// ---- HMI/VISUs/Templates/Motors/GUI_TEMPLATE_NOTT_MOTOR_CONTROL.TcVIS
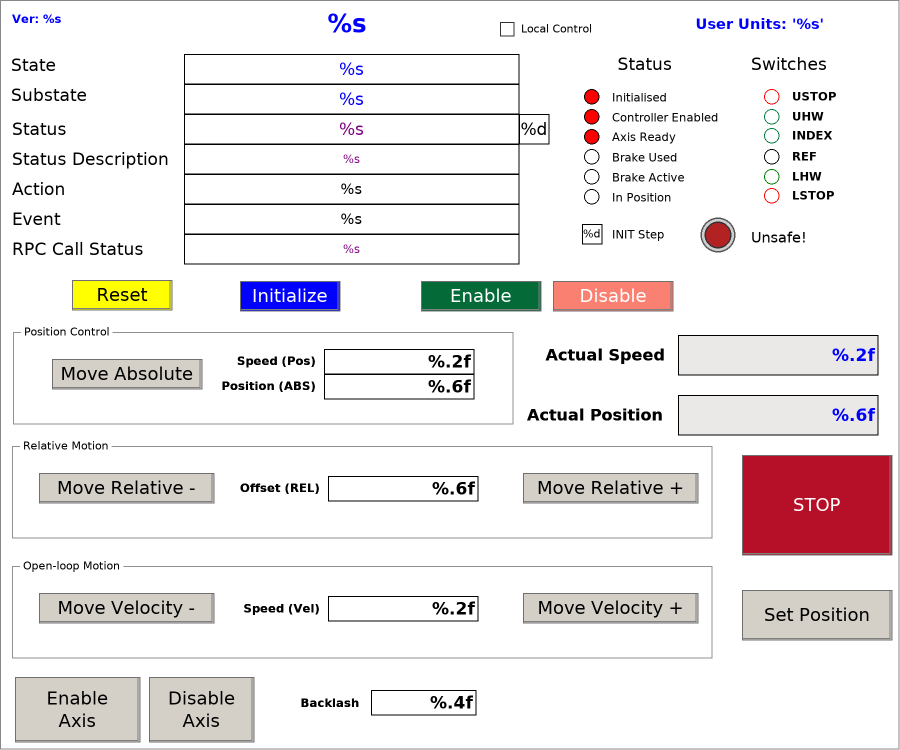
VISUALIZATION GUI_TEMPLATE_NOTT_MOTOR_CONTROL  // 900x750
VAR_IN_OUT
	m_Instance:	FB_NOTT_MOTOR;
END_VAR
VAR
	m_lrOffSet : LREAL := 0;
END_VAR
    GroupBox (12,558 700x100), "Open-loop Motion"
        Button (511,35 175x30), "Move Velocity +", input disabled if: NOT m_Instance.stat.bLocal OR NOT m_Instance.in_bSafe
            OnMouseDown: execute {
                m_Instance.ctrl.bLocalCmd := TRUE;
                m_Instance.ctrl.nCommand := E_MOTOR_COMMAND.MOTOR_MOVE;
                m_Instance.ctrl.nMoveType := E_MOTOR_MOVE_TYPE.VELOCITY;
                m_Instance.ctrl.nDirection := MC_Positive_Direction;
                m_Instance.ctrl.bExecute := TRUE;
            }
    Button (523,593 175x30), "Move Velocity +", input disabled if: NOT m_Instance.stat.bLocal OR NOT m_Instance.in_bSafe
        OnMouseDown: execute {
            m_Instance.ctrl.bLocalCmd := TRUE;
            m_Instance.ctrl.nCommand := E_MOTOR_COMMAND.MOTOR_MOVE;
            m_Instance.ctrl.nMoveType := E_MOTOR_MOVE_TYPE.VELOCITY;
            m_Instance.ctrl.nDirection := MC_Positive_Direction;
            m_Instance.ctrl.bExecute := TRUE;
        }
    GroupBox (12,438 700x100), "Relative Motion"
    GroupBox (13,324 500x100), "Position Control"
    Rectangle (184,54 335x30), "%s", text variable: m_Instance.stat.sState
    Rectangle (184,84 335x30), "%s", text variable: m_Instance.stat.sSubstate
    Button (72,280 100x30), "Reset", input disabled if: NOT m_Instance.stat.bLocal OR NOT m_Instance.in_bSafe
        OnMouseDown: execute {
            m_Instance.ctrl.bLocalCmd := TRUE;
            m_Instance.ctrl.nCommand := E_MOTOR_COMMAND.RESET;
            m_Instance.ctrl.bExecute := TRUE;
        }
    Button (240,281 100x30), "Initialize", input disabled if: NOT m_Instance.stat.bLocal OR NOT m_Instance.in_bSafe
        OnMouseDown: execute {
            m_Instance.ctrl.bLocalCmd := TRUE;
            m_Instance.ctrl.nCommand := E_MOTOR_COMMAND.INIT;
            m_Instance.ctrl.bExecute := TRUE;
        }
    Button (742,455 150x100), "STOP", input disabled if: NOT m_Instance.stat.bLocal OR NOT m_Instance.in_bSafe
        OnMouseDown: execute {
            m_Instance.ctrl.bLocalCmd := TRUE;
            m_Instance.ctrl.nCommand := E_MOTOR_COMMAND.STOP;
            m_Instance.ctrl.bExecute := TRUE;
        }
    Button (421,281 120x30), "Enable", input disabled if: NOT m_Instance.stat.bLocal OR NOT m_Instance.in_bSafe
        OnMouseDown: execute {
            m_Instance.ctrl.bLocalCmd := TRUE;
            m_Instance.ctrl.nCommand := E_MOTOR_COMMAND.ENABLE;
            m_Instance.ctrl.bExecute := TRUE;
        }
    Button (553,281 120x30), "Disable", input disabled if: NOT m_Instance.stat.bLocal OR NOT m_Instance.in_bSafe
        OnMouseDown: execute {
            m_Instance.ctrl.bLocalCmd := TRUE;
            m_Instance.ctrl.nCommand := E_MOTOR_COMMAND.DISABLE;
            m_Instance.ctrl.bExecute := TRUE;
        }
    Rectangle (8,50 170x30), "State"
    Rectangle (8,80 170x30), "Substate"
    Rectangle (184,114 335x30), "%s", text variable: m_Instance.stat.sStatus
    Rectangle (184,144 335x30), "%s", tooltip "Additional information mostly used for description of errors", text variable: m_Instance.stat.sErrorText
    Rectangle (9,114 170x30), "Status"
    Rectangle (9,144 170x30), "Status Description"
    Rectangle (184,174 335x30), "%s", text variable: m_Instance.stat.sActionDesc
    Rectangle (184,204 335x30), "%s", text variable: m_Instance.stat.sEventDesc
    Rectangle (9,174 170x30), "Action"
    Rectangle (9,204 170x30), "Event"
    Rectangle (231,6 232x35), "%s", text variable: m_Instance.sName
    Checkbox (498,14 116x30), "Local Control", variable: m_Instance.stat.bLocal
    Rectangle (599,49 92x30), "Status"
    Rectangle (519,114 30x30), "%d", text variable: m_Instance.stat.nStatus
    Rectangle (743,49 92x30), "Switches"
    Button (742,590 150x50), "Set Position", input disabled if: NOT m_Instance.stat.bLocal OR NOT m_Instance.in_bSafe
        OnMouseDown: execute {
            m_Instance.ctrl.bLocalCmd := TRUE;
            m_Instance.ctrl.nCommand := E_MOTOR_COMMAND.SET_POSITION;
            m_Instance.ctrl.bExecute := TRUE;
        }
    Rectangle (789,89 50x15), "USTOP"
    Ellipse (764,89 15x15), colour toggle: m_Instance.stat.signals[5].bActive
    Ellipse (764,109 15x15), colour toggle: m_Instance.stat.signals[4].bActive
    Ellipse (764,169 15x15), colour toggle: m_Instance.stat.signals[1].bActive
    Ellipse (764,188 15x15), colour toggle: m_Instance.stat.signals[0].bActive
    Ellipse (764,149 15x15), colour toggle: m_Instance.stat.signals[2].bActive
    Rectangle (789,128 50x15), "INDEX"
    Rectangle (789,109 50x15), "UHW"
    Rectangle (789,149 50x15), "REF"
    Rectangle (789,169 50x15), "LHW"
    Rectangle (789,188 50x15), "LSTOP"
    Ellipse (764,128 15x15), colour toggle: m_Instance.stat.signals[3].bActive
    Group (267,690 209x25)
        Rectangle (0,3 95x20), "Backlash"
        Rectangle (104,0 105x25), "%.4f", text variable: m_Instance.cfg.lrBacklash
            OnMouseDown: write the text variable via Default
    Rectangle (267,693 95x20), "Backlash"
    Rectangle (371,690 105x25), "%.4f", text variable: m_Instance.cfg.lrBacklash
        OnMouseDown: write the text variable via Default
    Button (52,359 150x30), "Move Absolute", input disabled if: NOT m_Instance.stat.bLocal OR NOT m_Instance.in_bSafe
        OnMouseDown: execute {
            m_Instance.ctrl.bLocalCmd := TRUE;
            m_Instance.ctrl.lrVelocity:=(m_Instance.cfg.lrDefaultVelocity);
            m_Instance.ctrl.nCommand := E_MOTOR_COMMAND.MOTOR_MOVE;
            m_Instance.ctrl.nMoveType := E_MOTOR_MOVE_TYPE.ABSOLUTE;
            m_Instance.ctrl.bExecute := TRUE;
        }
    Group (224,374 250x25)
        Rectangle (0,2 95x20), "Position (ABS)"
        Rectangle (100,0 150x25), "%.6f", tooltip "Absolute position used by "MOVE ABS"", text variable: m_Instance.ctrl.lrPosition
            OnMouseDown: write the text variable via Default
    Rectangle (224,376 95x20), "Position (ABS)"
    Rectangle (324,374 150x25), "%.6f", tooltip "Absolute position used by "MOVE ABS"", text variable: m_Instance.ctrl.lrPosition
        OnMouseDown: write the text variable via Default
    Group (224,349 250x25)
        Rectangle (0,2 95x20), "Speed (Pos)"
        Rectangle (100,0 150x25), "%.2f", text variable: m_Instance.cfg.lrDefaultVelocity
            OnMouseDown: write the text variable via Default
    Rectangle (224,351 95x20), "Speed (Pos)"
    Rectangle (324,349 150x25), "%.2f", text variable: m_Instance.cfg.lrDefaultVelocity
        OnMouseDown: write the text variable via Default
    Rectangle (609,165 90x25), "Brake Active"
    Ellipse (584,169 15x15), tooltip "RED = Applied BLANK = Released", colour toggle: (m_Instance.stat.bBrakeActive) <> 0
    Ellipse (584,89 15x15), tooltip "GREEN = Initialised RED = Not Initialised", text variable: m_Instance.stat.bInitialised, colour toggle: m_Instance.stat.bInitialised
    Rectangle (609,85 90x25), "Initialised"
    Rectangle (609,105 125x25), "Controller Enabled"
    Rectangle (609,125 90x24), "Axis Ready"
    Rectangle (609,145 90x25), "Brake Used"
    Ellipse (584,109 15x15), tooltip "GREEN = Enabled RED = Disabled", colour toggle: m_Instance.stat.bEnabled
    Ellipse (584,129 15x15), tooltip "GREEN = Ready RED = Not Ready", colour toggle: m_Instance.stat.bAxisReady
    Ellipse (584,149 15x15), tooltip "BLUE = Used BLANK = Not Used", colour toggle: m_Instance.cfg.bUseBrake
    Rectangle (582,224 20x20), "%d", text variable: m_Instance.stat.nInitStep
    Rectangle (609,222 90x25), "INIT Step"
    Rectangle (9,234 170x30), "RPC Call Status"
    Rectangle (184,234 335x30), "%s", text variable: m_Instance.stat.sRPCErrorText
    Rectangle (609,185 90x25), "In Position"
    Ellipse (584,189 15x15), tooltip "GREEN = In Position BLANK = Not In Position (or not used)", colour toggle: (m_Instance.stat.bInPosition) <> 0
    Button (15,677 125x65), "Enable Axis", input disabled if: NOT m_Instance.stat.bLocal OR NOT m_Instance.in_bSafe
        OnMouseDown: execute { m_Instance.stat.bEnabled := TRUE; }
    Button (149,677 105x65), "Disable Axis", input disabled if: NOT m_Instance.stat.bLocal OR NOT m_Instance.in_bSafe
        OnMouseDown: execute { m_Instance.stat.bEnabled := FALSE; }
    Rectangle (624,9 203x30), "User Units: '%s'", text variable: m_Instance.stat.axis.sUnits
    Rectangle (9,4 99x30), "Ver: %s", tooltip "'Motor.library version'", text variable: m_Instance.stat.sLibVersion, input disabled if: true
    Lamp1 (698,215 40x40), tooltip "If active, it is not safe to operate the motor.", variable: NOT m_Instance.in_bSafe, invisible if: m_Instance.in_bSafe, style: Lamp-Lamp1-Red
    Rectangle (738,227 82x21), "Unsafe!", invisible if: m_Instance.in_bSafe
    Group (518,335 360x40)
        Rectangle (160,0 200x40), "%.2f", text variable: m_Instance.stat.lrVelActual, input disabled if: false
        Rectangle (0,5 150x30), "Actual Speed"
    Rectangle (678,335 200x40), "%.2f", text variable: m_Instance.stat.lrVelActual, input disabled if: false
    Rectangle (518,340 150x30), "Actual Speed"
    Group (516,395 362x40)
        Rectangle (162,0 200x40), "%.6f", text variable: m_Instance.stat.lrPosActual, input disabled if: false
        Rectangle (0,5 150x30), "Actual Position"
    Rectangle (678,395 200x40), "%.6f", text variable: m_Instance.stat.lrPosActual, input disabled if: false
    Rectangle (516,400 150x30), "Actual Position"
    Group (228,596 250x25)
        Rectangle (0,0 95x25), "Speed (Vel)"
        Rectangle (100,0 150x25), "%.2f", text variable: m_Instance.ctrl.lrVelocity
            OnMouseDown: write the text variable via Default
    Rectangle (228,596 95x25), "Speed (Vel)"
    Rectangle (328,596 150x25), "%.2f", text variable: m_Instance.ctrl.lrVelocity
        OnMouseDown: write the text variable via Default
    Button (39,593 175x30), "Move Velocity -", input disabled if: NOT m_Instance.stat.bLocal OR NOT m_Instance.in_bSafe
        OnMouseDown: execute {
            m_Instance.ctrl.bLocalCmd := TRUE;
            m_Instance.ctrl.nCommand := E_MOTOR_COMMAND.MOTOR_MOVE;
            m_Instance.ctrl.nMoveType := E_MOTOR_MOVE_TYPE.VELOCITY;
            m_Instance.ctrl.nDirection := MC_Negative_Direction;
            m_Instance.ctrl.bExecute := TRUE;
        }
    Button (39,473 175x30), "Move Relative -", input disabled if: NOT m_Instance.stat.bLocal OR NOT m_Instance.in_bSafe
        OnMouseDown: execute {
            m_Instance.ctrl.bLocalCmd := TRUE;
            m_Instance.ctrl.lrOffset := m_lrOffSet * (-1);
            m_Instance.ctrl.lrVelocity:=(m_Instance.cfg.lrDefaultVelocity);
            m_Instance.ctrl.nCommand := E_MOTOR_COMMAND.MOTOR_MOVE;
            m_Instance.ctrl.nMoveType := E_MOTOR_MOVE_TYPE.RELATIVE;
            m_Instance.ctrl.bExecute := TRUE;
        }
    Group (228,476 250x25)
        Rectangle (0,2 95x20), "Offset (REL)"
        Rectangle (100,0 150x25), "%.6f", tooltip "Relative offset used by "MOVE REL"", text variable: m_lrOffSet
            OnMouseDown: write the text variable via Default
    Rectangle (228,478 95x20), "Offset (REL)"
    Rectangle (328,476 150x25), "%.6f", tooltip "Relative offset used by "MOVE REL"", text variable: m_lrOffSet
        OnMouseDown: write the text variable via Default
    Button (523,473 175x30), "Move Relative +", input disabled if: NOT m_Instance.stat.bLocal OR NOT m_Instance.in_bSafe
        OnMouseDown: execute {
            m_Instance.ctrl.bLocalCmd := TRUE;
            m_Instance.ctrl.lrOffset := m_lrOffSet;
            m_Instance.ctrl.lrVelocity:=(m_Instance.cfg.lrDefaultVelocity);
            m_Instance.ctrl.nCommand := E_MOTOR_COMMAND.MOTOR_MOVE;
            m_Instance.ctrl.nMoveType := E_MOTOR_MOVE_TYPE.RELATIVE;
            m_Instance.ctrl.bExecute := TRUE;
        }
END_VISUALIZATION

// ---- HMI/VISUs/Templates/Shutters/GUI_TEMPLATE_NOTT_SHUTTER.TcVIS
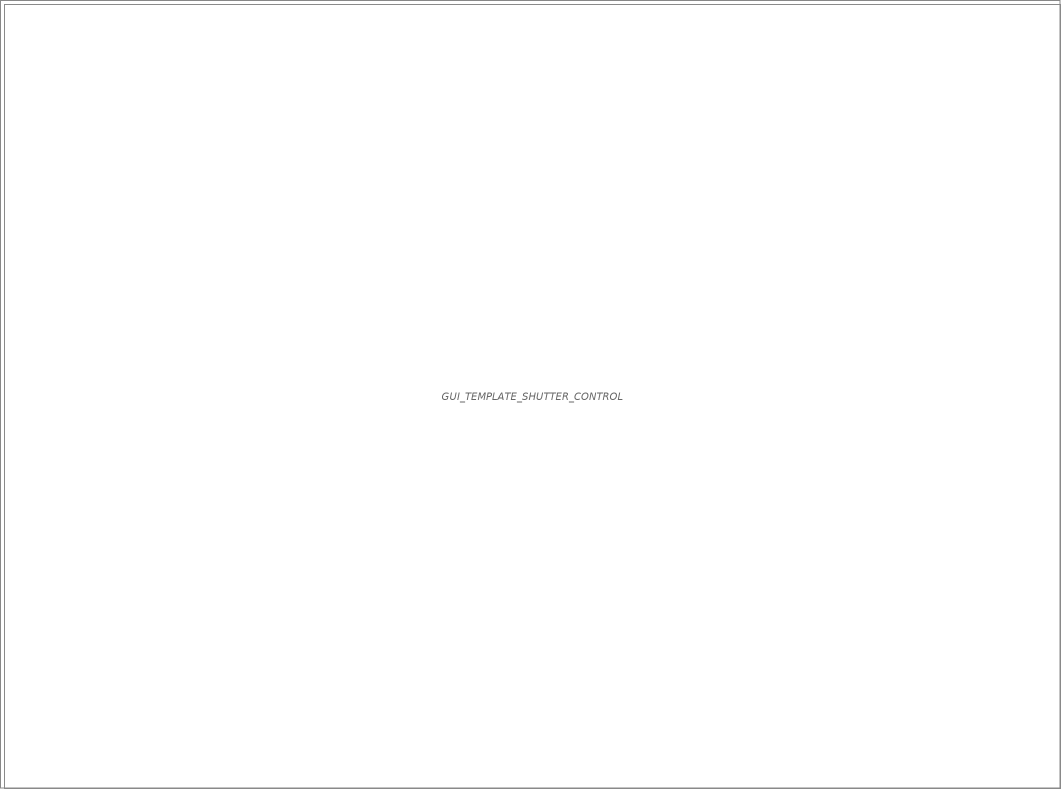
VISUALIZATION GUI_TEMPLATE_NOTT_SHUTTER  // 1061x789
VAR_IN_OUT
	m_Instance:	FB_NOTT_MOTOR;
END_VAR
    TabControl (4,4 1057x785)
        shows GUI_TEMPLATE_SHUTTER_CONTROL(m_Instance := m_Instance)
        shows GUI_TEMPLATE_NOTT_MOTOR_CONFIG(m_Instance := m_Instance)
        [0]: TabTitle=Shutter Control
        [1]: TabTitle=Config
END_VISUALIZATION

// ---- HMI/VISUs/Templates/Shutters/GUI_TEMPLATE_SHUTTER_CONTROL.TcVIS
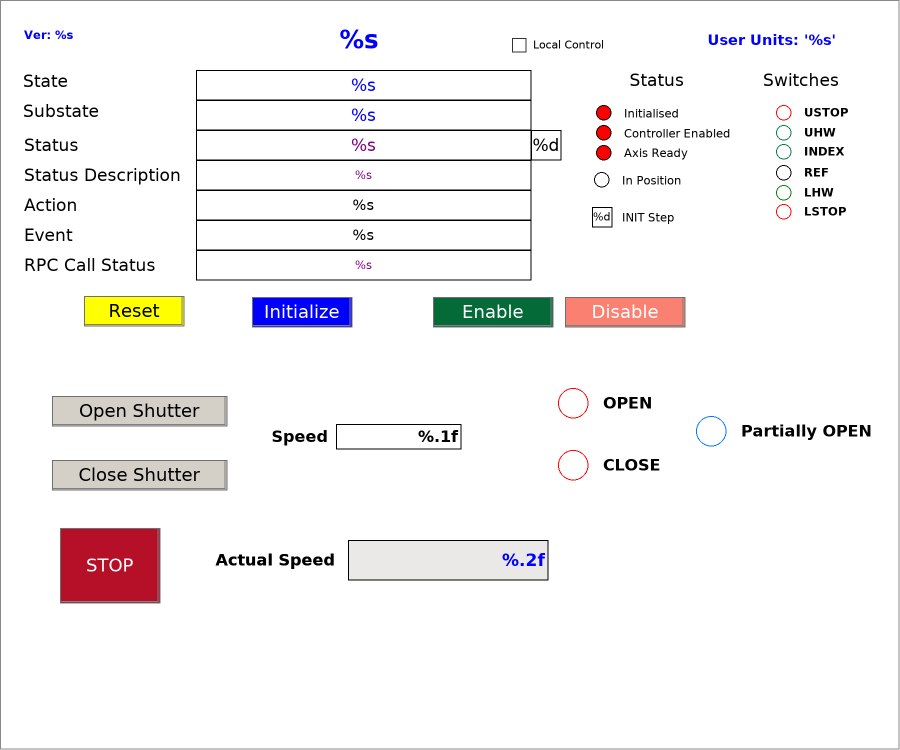
VISUALIZATION GUI_TEMPLATE_SHUTTER_CONTROL  // 900x750
VAR_IN_OUT
	m_Instance:	FB_NOTT_MOTOR;
END_VAR
VAR
	m_lrOffSet : LREAL := 0;
END_VAR
    Rectangle (196,70 335x30), "%s", text variable: m_Instance.stat.sState
    Rectangle (196,100 335x30), "%s", text variable: m_Instance.stat.sSubstate
    Button (84,296 100x30), "Reset", input disabled if: NOT m_Instance.stat.bLocal OR NOT m_Instance.in_bSafe
        OnMouseDown: execute {
            m_Instance.ctrl.bLocalCmd := TRUE;
            m_Instance.ctrl.nCommand := E_MOTOR_COMMAND.RESET;
            m_Instance.ctrl.bExecute := TRUE;
        }
    Button (252,297 100x30), "Initialize", input disabled if: NOT m_Instance.stat.bLocal OR NOT m_Instance.in_bSafe
        OnMouseDown: execute {
            m_Instance.ctrl.bLocalCmd := TRUE;
            m_Instance.ctrl.nCommand := E_MOTOR_COMMAND.INIT;
            m_Instance.ctrl.bExecute := TRUE;
        }
    Button (60,528 100x75), "STOP", input disabled if: NOT m_Instance.stat.bLocal OR NOT m_Instance.in_bSafe
        OnMouseDown: execute {
            m_Instance.ctrl.bLocalCmd := TRUE;
            m_Instance.ctrl.nCommand := E_MOTOR_COMMAND.STOP;
            m_Instance.ctrl.bExecute := TRUE;
        }
    Button (433,297 120x30), "Enable", input disabled if: NOT m_Instance.stat.bLocal OR NOT m_Instance.in_bSafe
        OnMouseDown: execute {
            m_Instance.ctrl.bLocalCmd := TRUE;
            m_Instance.ctrl.nCommand := E_MOTOR_COMMAND.ENABLE;
            m_Instance.ctrl.bExecute := TRUE;
        }
    Button (565,297 120x30), "Disable", input disabled if: NOT m_Instance.stat.bLocal OR NOT m_Instance.in_bSafe
        OnMouseDown: execute {
            m_Instance.ctrl.bLocalCmd := TRUE;
            m_Instance.ctrl.nCommand := E_MOTOR_COMMAND.DISABLE;
            m_Instance.ctrl.bExecute := TRUE;
        }
    Rectangle (20,66 170x30), "State"
    Rectangle (20,96 170x30), "Substate"
    Rectangle (196,130 335x30), "%s", text variable: m_Instance.stat.sStatus
    Rectangle (196,160 335x30), "%s", tooltip "Additional information mostly used for description of errors", text variable: m_Instance.stat.sErrorText
    Rectangle (21,130 170x30), "Status"
    Rectangle (21,160 170x30), "Status Description"
    Rectangle (196,190 335x30), "%s", text variable: m_Instance.stat.sActionDesc
    Rectangle (196,220 335x30), "%s", text variable: m_Instance.stat.sEventDesc
    Rectangle (21,190 170x30), "Action"
    Rectangle (21,220 170x30), "Event"
    Rectangle (243,22 232x35), "%s", text variable: m_Instance.sName
    Checkbox (510,30 116x30), "Local Control", variable: m_Instance.stat.bLocal
    Rectangle (611,65 92x30), "Status"
    Rectangle (531,130 30x30), "%d", text variable: m_Instance.stat.nStatus
    Rectangle (755,65 92x30), "Switches"
    Rectangle (801,105 50x15), "USTOP"
    Ellipse (776,105 15x15), colour toggle: m_Instance.stat.signals[5].bActive
    Ellipse (776,125 15x15), colour toggle: m_Instance.stat.signals[4].bActive
    Ellipse (776,185 15x15), colour toggle: m_Instance.stat.signals[1].bActive
    Ellipse (776,204 15x15), colour toggle: m_Instance.stat.signals[0].bActive
    Ellipse (776,165 15x15), colour toggle: m_Instance.stat.signals[2].bActive
    Rectangle (801,144 50x15), "INDEX"
    Rectangle (801,125 50x15), "UHW"
    Rectangle (801,165 50x15), "REF"
    Rectangle (801,185 50x15), "LHW"
    Rectangle (801,204 50x15), "LSTOP"
    Ellipse (776,144 15x15), colour toggle: m_Instance.stat.signals[3].bActive
    Ellipse (596,105 15x15), tooltip "GREEN = Initialised RED = Not Initialised", text variable: m_Instance.stat.bInitialised, colour toggle: m_Instance.stat.bInitialised
    Rectangle (621,101 90x25), "Initialised"
    Rectangle (621,121 125x25), "Controller Enabled"
    Rectangle (621,141 90x24), "Axis Ready"
    Ellipse (596,125 15x15), tooltip "GREEN = Enabled RED = Disabled", colour toggle: m_Instance.stat.bEnabled
    Ellipse (596,145 15x15), tooltip "GREEN = Ready RED = Not Ready", colour toggle: m_Instance.stat.bAxisReady
    Rectangle (592,207 20x20), "%d", text variable: m_Instance.stat.nInitStep
    Rectangle (619,205 90x25), "INIT Step"
    Rectangle (21,250 170x30), "RPC Call Status"
    Rectangle (196,250 335x30), "%s", text variable: m_Instance.stat.sRPCErrorText
    Rectangle (619,168 90x25), "In Position"
    Ellipse (594,172 15x15), tooltip "GREEN = In Position BLANK = Not In Position (or not used)", colour toggle: (m_Instance.stat.bInPosition) <> 0
    Rectangle (636,25 203x30), "User Units: '%s'", text variable: m_Instance.stat.axis.sUnits
    Rectangle (21,20 99x30), "Ver: %s", tooltip "'Motor.library version'", text variable: m_Instance.stat.sLibVersion, input disabled if: true
    Group (188,540 360x40)
        Rectangle (160,0 200x40), "%.2f", text variable: m_Instance.stat.lrVelActual, input disabled if: false
        Rectangle (0,5 150x30), "Actual Speed"
    Rectangle (348,540 200x40), "%.2f", text variable: m_Instance.stat.lrVelActual, input disabled if: false
    Rectangle (188,545 150x30), "Actual Speed"
    Rectangle (236,424 95x25), "Speed", tooltip "Shutter Speed (mm/sec)"
    Rectangle (336,424 125x25), "%.1f", text variable: m_Instance.ctrl.lrVelocity
        OnMouseDown: write the text variable via Default
    Button (52,396 175x30), "Open Shutter", input disabled if: NOT m_Instance.stat.bLocal OR NOT m_Instance.in_bSafe
        OnMouseDown: execute {
            m_Instance.ctrl.bLocalCmd := TRUE;
            m_Instance.ctrl.nCommand := E_MOTOR_COMMAND.MOTOR_MOVE;
            m_Instance.ctrl.nMoveType := E_MOTOR_MOVE_TYPE.VELOCITY;
            m_Instance.ctrl.nDirection := MC_Negative_Direction;
            m_Instance.ctrl.bExecute := TRUE;
        }
    Button (52,460 175x30), "Close Shutter", input disabled if: NOT m_Instance.stat.bLocal OR NOT m_Instance.in_bSafe
        OnMouseDown: execute {
            m_Instance.ctrl.bLocalCmd := TRUE;
            m_Instance.ctrl.nCommand := E_MOTOR_COMMAND.MOTOR_MOVE;
            m_Instance.ctrl.nMoveType := E_MOTOR_MOVE_TYPE.VELOCITY;
            m_Instance.ctrl.nDirection := MC_Positive_Direction;
            m_Instance.ctrl.bExecute := TRUE;
        }
    Ellipse (558,388 30x30), colour toggle: m_Instance.stat.signals[0].bActive
    Rectangle (600,388 100x30), "OPEN", tooltip "Shutter is Open"
    Ellipse (558,450 30x30), colour toggle: m_Instance.stat.signals[5].bActive
    Rectangle (600,450 100x30), "CLOSE", tooltip "Shutter is closed"
    Ellipse (696,416 30x30), colour toggle: m_Instance.bShutterPartiallyOpen
    Rectangle (738,416 143x30), "Partially OPEN", tooltip "Either shutter is opening or closing"
END_VISUALIZATION

// ---- HMI/VISUs/Util/Button/VISU_HMI_ROUTINES_BUTTON.TcVIS
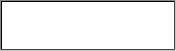
VISUALIZATION VISU_HMI_ROUTINES_BUTTON  // 176x51
VAR_IN_OUT
    m_Hmi : FB_HMI_BUTTON;
END_VAR
    Rectangle (0,0 175x50), invisible if: m_Hmi.bIsNotOrange
    Rectangle (0,0 175x50), invisible if: m_Hmi.bIsNotGray
    Rectangle (0,0 175x50), invisible if: m_Hmi.bIsNotBlue
    Rectangle (0,0 175x50), invisible if: m_Hmi.bIsNotRed
    Rectangle (0,0 175x50), invisible if: m_Hmi.bIsNotGreen
    Rectangle (0,0 175x50), "%s", text variable: m_Hmi.sName
    Rectangle (0,0 175x50), invisible if: m_Hmi.bNotActivated
    Line (0,49) (175,49), invisible if: m_Hmi.bActivated
    Line (174,0) (174,50), invisible if: m_Hmi.bActivated
    Line (174,0) (0,0), invisible if: m_Hmi.bActivated
    Line (0,49) (0,0), invisible if: m_Hmi.bActivated
    Line (175,50) (175,1), invisible if: m_Hmi.bNotActivated
    Line (0,1) (174,1), invisible if: m_Hmi.bNotActivated
    Line (1,0) (1,49), invisible if: m_Hmi.bNotActivated
    Line (175,50) (1,50), invisible if: m_Hmi.bNotActivated
END_VISUALIZATION

// ---- HMI/VISUs/Util/Button/VISU_HMI_SUBSUBSYSTEM_BUTTON.TcVIS
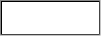
VISUALIZATION VISU_HMI_SUBSUBSYSTEM_BUTTON  // 101x36
VAR_IN_OUT
    m_Hmi : FB_HMI_BUTTON;
END_VAR
    Rectangle (0,0 100x35), invisible if: m_Hmi.bIsNotOrange
    Rectangle (0,0 100x35), invisible if: m_Hmi.bIsNotGray
    Rectangle (0,0 100x35), invisible if: m_Hmi.bIsNotBlue
    Rectangle (0,0 100x35), invisible if: m_Hmi.bIsNotRed
    Rectangle (0,0 100x35), invisible if: m_Hmi.bIsNotGreen
    Rectangle (0,0 100x35), "%s", text variable: m_Hmi.sName
    Rectangle (0,0 100x35), invisible if: m_Hmi.bNotActivated
    Line (0,34) (100,34), invisible if: m_Hmi.bActivated
    Line (99,0) (99,35), invisible if: m_Hmi.bActivated
    Line (98,0) (0,0), invisible if: m_Hmi.bActivated
    Line (0,35) (0,0), invisible if: m_Hmi.bActivated
    Line (100,35) (100,1), invisible if: m_Hmi.bNotActivated
    Line (0,1) (99,1), invisible if: m_Hmi.bNotActivated
    Line (1,0) (1,35), invisible if: m_Hmi.bNotActivated
    Line (100,35) (1,35), invisible if: m_Hmi.bNotActivated
END_VISUALIZATION

// ---- HMI/VISUs/Util/Button/VISU_HMI_SUBSYSTEM_BUTTON.TcVIS
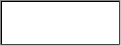
VISUALIZATION VISU_HMI_SUBSYSTEM_BUTTON  // 121x46
VAR_IN_OUT
    m_Hmi : FB_HMI_BUTTON;
END_VAR
    Rectangle (0,0 120x45), invisible if: m_Hmi.bIsNotOrange
    Rectangle (0,0 120x45), invisible if: m_Hmi.bIsNotGray
    Rectangle (0,0 120x45), invisible if: m_Hmi.bIsNotBlue
    Rectangle (0,0 120x45), invisible if: m_Hmi.bIsNotRed
    Rectangle (0,0 120x45), invisible if: m_Hmi.bIsNotGreen
    Rectangle (0,0 120x45), "%s", text variable: m_Hmi.sName
    Rectangle (0,0 120x45), invisible if: m_Hmi.bNotActivated
    Line (0,44) (120,44), invisible if: m_Hmi.bActivated
    Line (119,0) (119,45), invisible if: m_Hmi.bActivated
    Line (118,0) (0,0), invisible if: m_Hmi.bActivated
    Line (0,45) (0,0), invisible if: m_Hmi.bActivated
    Line (120,45) (120,1), invisible if: m_Hmi.bNotActivated
    Line (0,1) (119,1), invisible if: m_Hmi.bNotActivated
    Line (1,0) (1,45), invisible if: m_Hmi.bNotActivated
    Line (120,45) (1,45), invisible if: m_Hmi.bNotActivated
END_VISUALIZATION

// ---- HMI/VISUs/Util/Button/VISU_HMI_SYSTEM_BUTTON.TcVIS
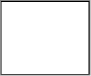
VISUALIZATION VISU_HMI_SYSTEM_BUTTON  // 91x76
VAR_IN_OUT
    m_Hmi : FB_HMI_BUTTON;
END_VAR
    Rectangle (0,0 90x75), invisible if: m_Hmi.bIsNotOrange
    Rectangle (0,0 90x75), invisible if: m_Hmi.bIsNotGray
    Rectangle (0,0 90x75), invisible if: m_Hmi.bIsNotBlue
    Rectangle (0,0 90x75), invisible if: m_Hmi.bIsNotRed
    Rectangle (0,0 90x75), invisible if: m_Hmi.bIsNotGreen
    Rectangle (0,50 90x25), "%s", text variable: m_Hmi.sName
    Image (25,10 40x40), image: VISU_HMI_BUTTON_IMAGES.Start
        p84334746: m_Hmi.sIconName
    Rectangle (0,0 90x75), invisible if: m_Hmi.bNotActivated
    Line (0,74) (90,74), invisible if: m_Hmi.bActivated
    Line (89,75) (89,0), invisible if: m_Hmi.bActivated
    Line (0,74) (0,0), invisible if: m_Hmi.bActivated
    Line (88,0) (0,0), invisible if: m_Hmi.bActivated
    Line (0,1) (90,1), invisible if: m_Hmi.bNotActivated
    Line (1,75) (1,0), invisible if: m_Hmi.bNotActivated
    Line (90,75) (1,75), invisible if: m_Hmi.bNotActivated
    Line (90,75) (90,1), invisible if: m_Hmi.bNotActivated
END_VISUALIZATION

// ---- HMI/VISU_HMI.TcVIS
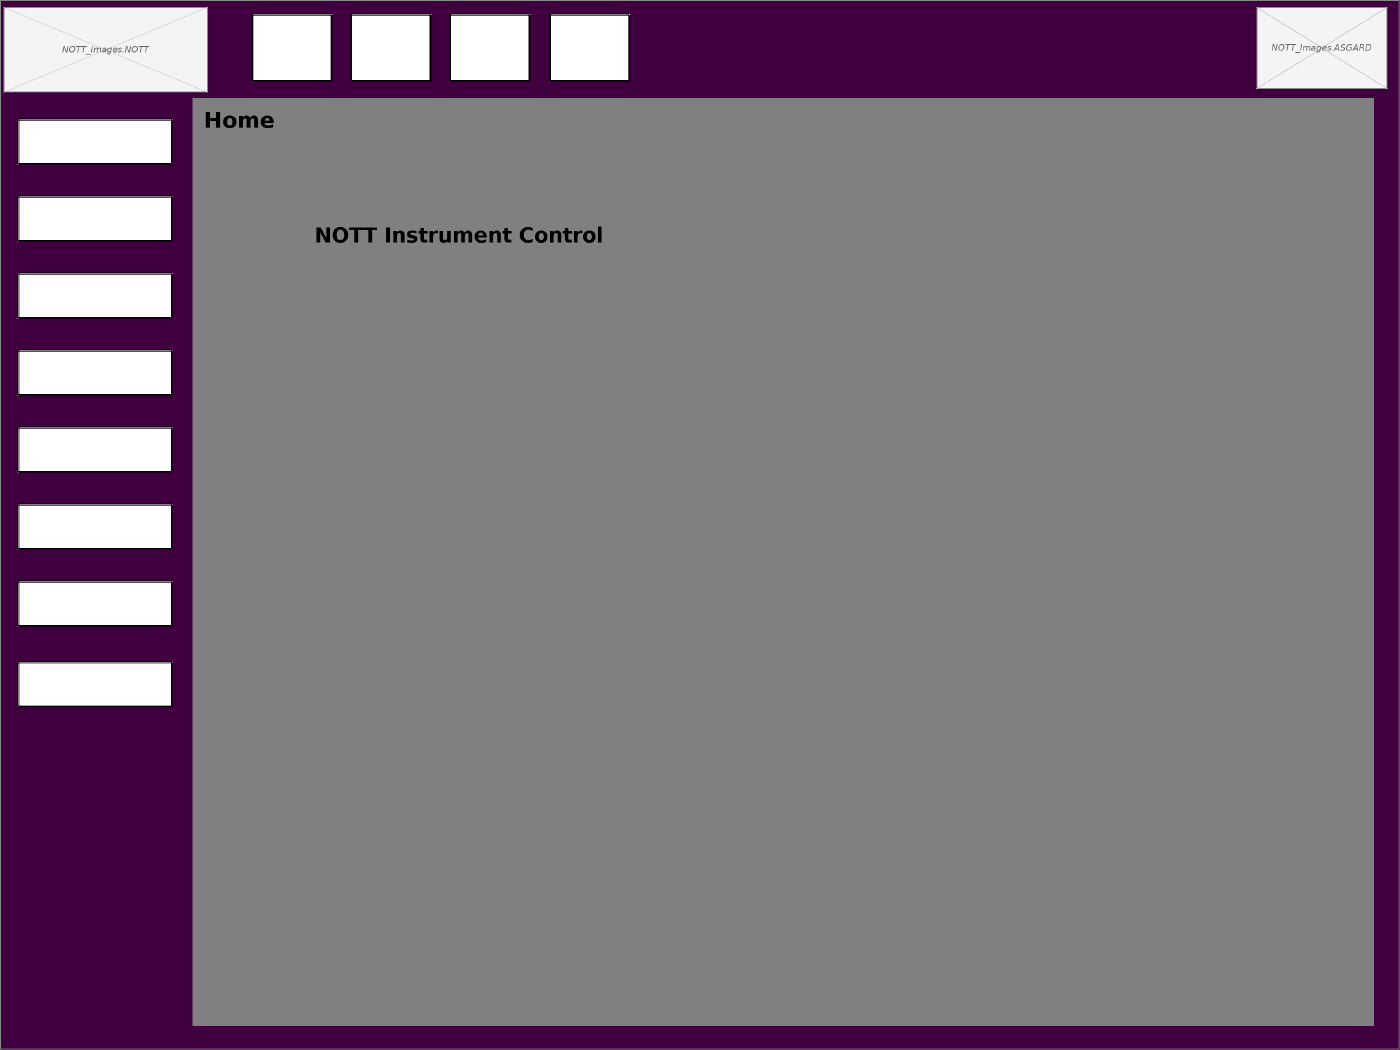
VISUALIZATION VISU_HMI  // 1600x1200
    Rectangle (220,112 1350x1060)
    Frame (220,112 1350x1060), frame switch variable: PRG_HMI.eActiveTab
        shows VISU_HMI_HOME(m_instance := MAIN.nott_ics)
        shows VISU_HMI_SERVICES(m_Instance := MAIN.fbServices)
        shows VISU_HMI_EVENTS()
        shows VISU_HMI_CRYO_INTERLOCKS()
        shows VISU_HMI_SHUTTERS()
        shows VISU_HMI_TIP_TILT(m_Hmi := PRG_HMI.fbTipTilt)
        shows VISU_HMI_DELAY_LINES()
        shows VISU_HMI_CO2_TRANS_STAGES()
        shows VISU_HMI_ZNSE_ACTUATORS()
        shows VISU_HMI_BIREFRINGENCE()
        shows VISU_HMI_BEAM_SPLITTER()
        shows VISU_HMI_CO2_PRESSURE()
        shows VISU_HMI_CRY(met_cryo_ctrl := MAIN.met_cryo_ctrl, m_Hmi := PRG_HMI.fbCry)
        shows VISU_HMI_CFO()
        shows VISU_HMI_IMG(m_Temperatures := MAIN.met_cryo_ctrl.met_temp, m_Voters := MAIN.met_cryo_ctrl.met_voters, m_Tctrl := MAIN.met_cryo_ctrl.met_tctrl, m_Heaters := MAIN.met_cryo_ctrl.met_heaters, m_Lakeshores := MAIN.met_cryo_ctrl.met_lakeshores, m_Hmi := PRG_HMI.fbImg)
        shows VISU_HMI_LMS()
        shows VISU_HMI_SCA(m_Temperatures := MAIN.met_cryo_ctrl.met_temp, m_Voters := MAIN.met_cryo_ctrl.met_voters, m_Tctrl := MAIN.met_cryo_ctrl.met_tctrl, m_Heaters := MAIN.met_cryo_ctrl.met_heaters, m_Lakeshores := MAIN.met_cryo_ctrl.met_lakeshores, m_Hmi := PRG_HMI.fbSca)
        shows VISU_HMI_HEATERS()
        shows VISU_HMI_EVENTS()
        shows VISU_HMI_PRESSURES()
        shows VISU_HMI_COOLERS()
        shows VISU_HMI_PUMPS(m_Hmi := PRG_HMI.fbPumps)
        shows VISU_HMI_TEMPERATURES(met_cryo_ctrl := MAIN.met_cryo_ctrl, m_Hmi := PRG_HMI.fbTemperatures)
        shows VISU_HMI_ICS_INTERLOCKS()
        shows VISU_HMI_DETECTORS()
        shows VISU_HMI_CONTROL_LOOPS()
        p1199675002: PRG_HMI.fbSca
        p1171169602: PRG_HMI.fbPumps
    Frame (288,16 93x78)
        shows VISU_HMI_SYSTEM_BUTTON(m_Hmi := PRG_HMI.fbHomeButton)
        OnMouseClick: execute { PRG_HMI.eActiveTab := E_HMI_TABS.HOME; }
    Frame (401,16 93x78)
        shows VISU_HMI_SYSTEM_BUTTON(m_Hmi := PRG_HMI.fbServicesButton)
        OnMouseClick: execute { PRG_HMI.eActiveTab := E_HMI_TABS.SERVICES; }
    Frame (514,16 93x78)
        shows VISU_HMI_SYSTEM_BUTTON(m_Hmi := PRG_HMI.fbEventsButton)
        OnMouseClick: execute { PRG_HMI.eActiveTab := E_HMI_TABS.EVENTS; }
    Frame (628,16 93x78)
        shows VISU_HMI_SYSTEM_BUTTON(m_Hmi := PRG_HMI.fbCryoInterlocksButton)
        OnMouseClick: execute { PRG_HMI.eActiveTab := E_HMI_TABS.CRYO_INTERLOCKS; }
    Frame (20,136 178x53)
        shows VISU_HMI_ROUTINES_BUTTON(m_Hmi := PRG_HMI.fbShuttersButton)
        OnMouseClick: execute { PRG_HMI.eActiveTab := E_HMI_TABS.SHUTTERS; }
    Frame (20,224 178x53)
        shows VISU_HMI_ROUTINES_BUTTON(m_Hmi := PRG_HMI.fbTipTiltButton)
        OnMouseClick: execute { PRG_HMI.eActiveTab := E_HMI_TABS.TIP_TILT; }
    Frame (20,312 178x53)
        shows VISU_HMI_ROUTINES_BUTTON(m_Hmi := PRG_HMI.fbDelayLinesButton)
        OnMouseClick: execute { PRG_HMI.eActiveTab := E_HMI_TABS.DELAY_LINES; }
    Frame (20,400 178x53)
        shows VISU_HMI_ROUTINES_BUTTON(m_Hmi := PRG_HMI.fbCO2TransStagesButton)
        OnMouseClick: execute { PRG_HMI.eActiveTab := E_HMI_TABS.CO2_TRANSLATION_STAGES; }
    Frame (20,488 178x53)
        shows VISU_HMI_ROUTINES_BUTTON(m_Hmi := PRG_HMI.fbZnSeActuatorsButton)
        OnMouseClick: execute { PRG_HMI.eActiveTab := E_HMI_TABS.ZNSE_ACTUATORS; }
    Frame (20,576 178x53)
        shows VISU_HMI_ROUTINES_BUTTON(m_Hmi := PRG_HMI.fbBirefringenceButton)
        OnMouseClick: execute { PRG_HMI.eActiveTab := E_HMI_TABS.BIREFRINGENCE_ACTUATORS; }
    Frame (20,664 178x53)
        shows VISU_HMI_ROUTINES_BUTTON(m_Hmi := PRG_HMI.fbBeamSplitterButton)
        OnMouseClick: execute { PRG_HMI.eActiveTab := E_HMI_TABS.CALIBRATION_UNIT_BEAM_SPLITER; }
    Frame (20,756 178x53)
        shows VISU_HMI_ROUTINES_BUTTON(m_Hmi := PRG_HMI.fbCO2PressureButton)
        OnMouseClick: execute { PRG_HMI.eActiveTab := E_HMI_TABS.CO2_PRESSURE_CONTROL; }
    Image (4,8 233x97), image: NOTT_Images.NOTT
    Image (1436,8 149x93), image: NOTT_Images.ASGARD
END_VISUALIZATION

// ---- VISUs/GUIs/Cryo/GUI_CRYO_TEMPS.TcVIS
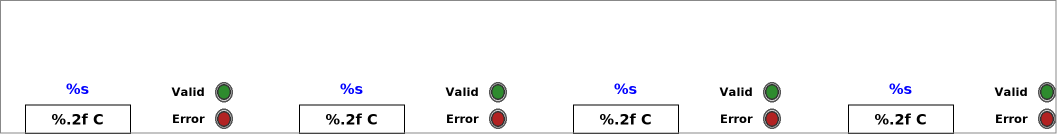
VISUALIZATION GUI_CRYO_TEMPS  // 1057x134
    Frame (9,56 225x78)
        shows TEMPLATE_NOTT_CRYO_TEMPS(m_instance := MAIN.not_cryo_ctrl.temp_1)
    Frame (283,56 225x78)
        shows TEMPLATE_NOTT_CRYO_TEMPS(m_instance := MAIN.not_cryo_ctrl.temp_2)
    Frame (557,56 225x78)
        shows TEMPLATE_NOTT_CRYO_TEMPS(m_instance := MAIN.not_cryo_ctrl.temp_3)
    Frame (832,56 225x78)
        shows TEMPLATE_NOTT_CRYO_TEMPS(m_instance := MAIN.not_cryo_ctrl.temp_4)
END_VISUALIZATION

// ---- VISUs/GUIs/NBS/GUI_NOTT_NBS.TcVIS
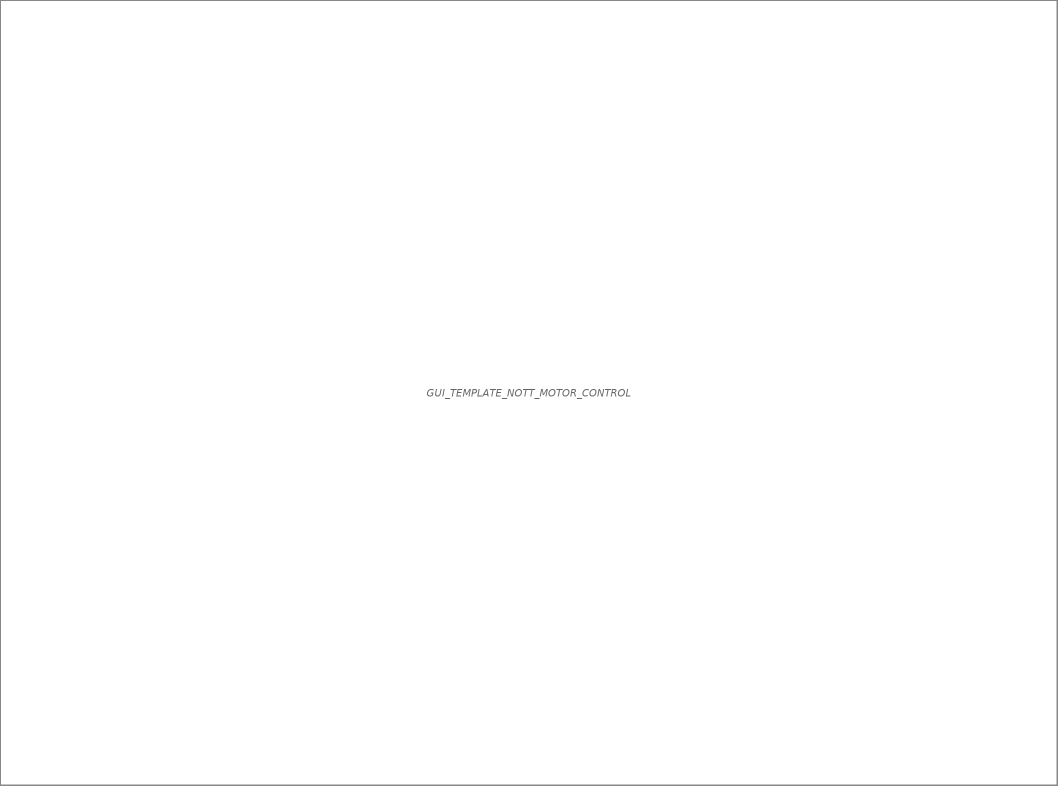
VISUALIZATION GUI_NOTT_NBS  // 1058x786
    Frame (0,0 1058x786)
        shows GUI_TEMPLATE_MOTOR(m_Instance := MAIN.nott_ics.Calibration_Unit_Beam_Splitter.NBS)
END_VISUALIZATION

// ---- VISUs/GUIs/Shutters/GUI_TEST_STEPPER_SHUTTER.TcVIS
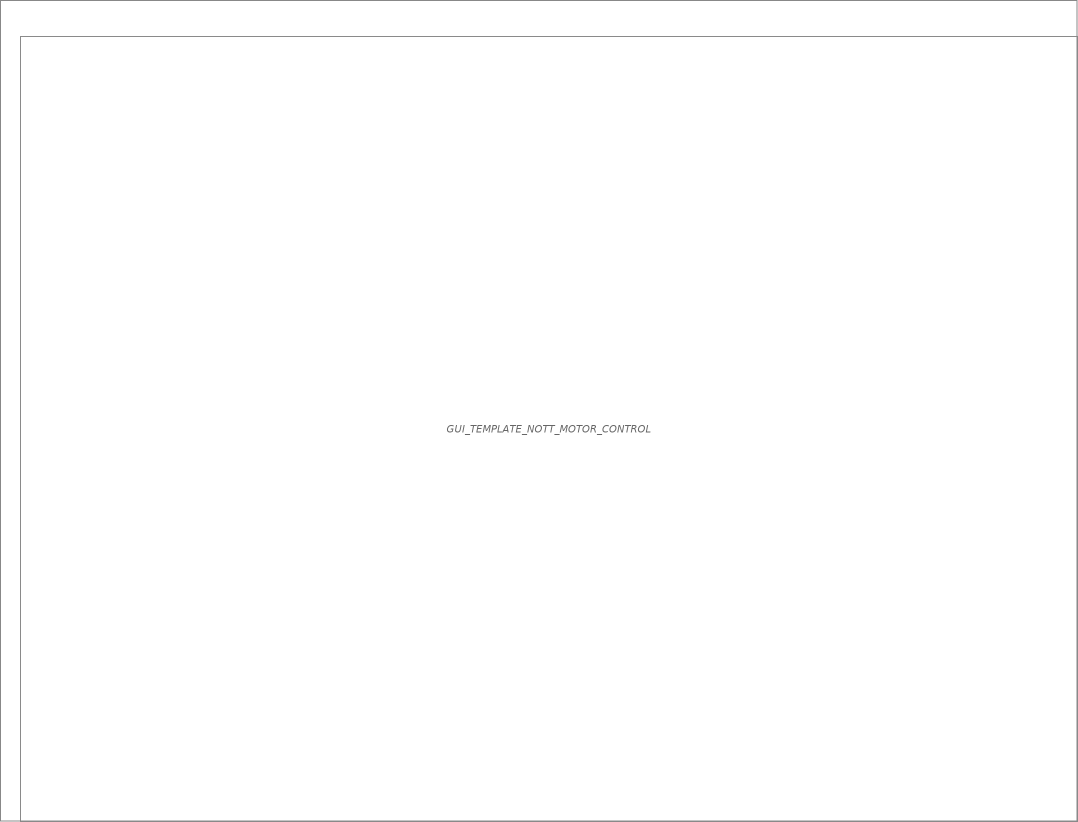
VISUALIZATION GUI_TEST_STEPPER_SHUTTER  // 1078x822
    Frame (20,36 1058x786)
        shows GUI_TEMPLATE_MOTOR(m_Instance := MAIN.nott_ics.Shutters.Test_Shutter)
END_VISUALIZATION

// ---- VISUs/GUIs/Templates/TEMPLATE_NOTT_CRYO_TEMPS.TcVIS
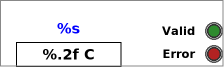
VISUALIZATION TEMPLATE_NOTT_CRYO_TEMPS  // 224x67
VAR_IN_OUT
	m_instance:		FB_CRYO_SENSOR_TEMPERATURE;
END_VAR
    Rectangle (16,16 105x25), "%s", text variable: m_instance.in_sName
    Rectangle (16,42 105x25), "%.2f C", tooltip "Temperature in C", text variable: m_instance.stat.lrTempC
        OnMouseDown: write the text variable via Default
    Group (138,21 86x20)
        Lamp1 (66,0 20x20), variable: m_instance.stat.bValid, style: Lamp-Lamp1-Green
        Rectangle (0,0 60x20), "Valid"
    Group (138,44 86x20)
        Lamp1 (66,0 20x20), variable: m_instance.stat.bError, style: Lamp-Lamp1-Red
        Rectangle (0,0 60x20), "Error"
END_VISUALIZATION

// ---- VISUs/GUIs/Delay_Lines/GUI_NOTT_DL_CONFIG.TcVIS
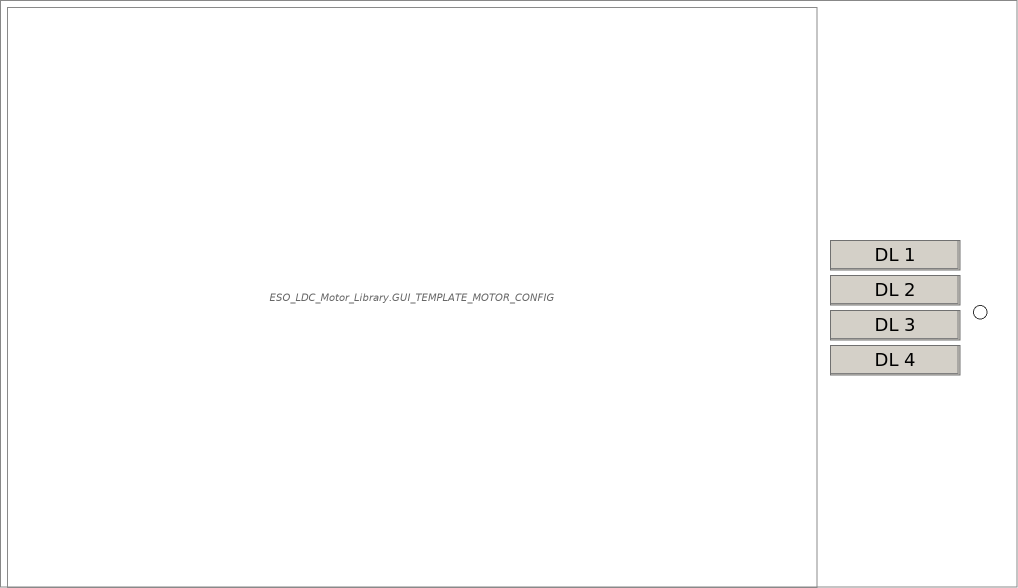
VISUALIZATION GUI_NOTT_DL_CONFIG  // 1018x588
    RadioButton (971,242 47x140), variable: MAIN.nott_ics.Delay_Lines.guiShutterIndex-1
        Areas[0]: Text=Radiobutton
        Areas[1]: Text=Radiobutton
    Button (830,240 130x30), "DL 1"
        OnMouseClick: execute { MAIN.nott_ics.Delay_Lines.guiShutterIndex := 1; }
    Button (830,275 130x30), "DL 2"
        OnMouseClick: execute { MAIN.nott_ics.Delay_Lines.guiShutterIndex := 2; }
    Button (830,310 130x30), "DL 3"
        OnMouseClick: execute { MAIN.nott_ics.Delay_Lines.guiShutterIndex := 3; }
    Button (830,345 130x30), "DL 4"
        OnMouseClick: execute { MAIN.nott_ics.Delay_Lines.guiShutterIndex := 4; }
    Frame (7,7 810x581)
        shows ESO_LDC_Motor_Library.GUI_TEMPLATE_MOTOR_CONFIG(m_Instance := MAIN.nott_ics.Delay_Lines.ptrDelayLines[MAIN.nott_ics.Delay_Lines.guiShutterIndex]^)
END_VISUALIZATION

// ---- VISUs/GUIs/Delay_Lines/GUI_NOTT_DL_CTRL.TcVIS
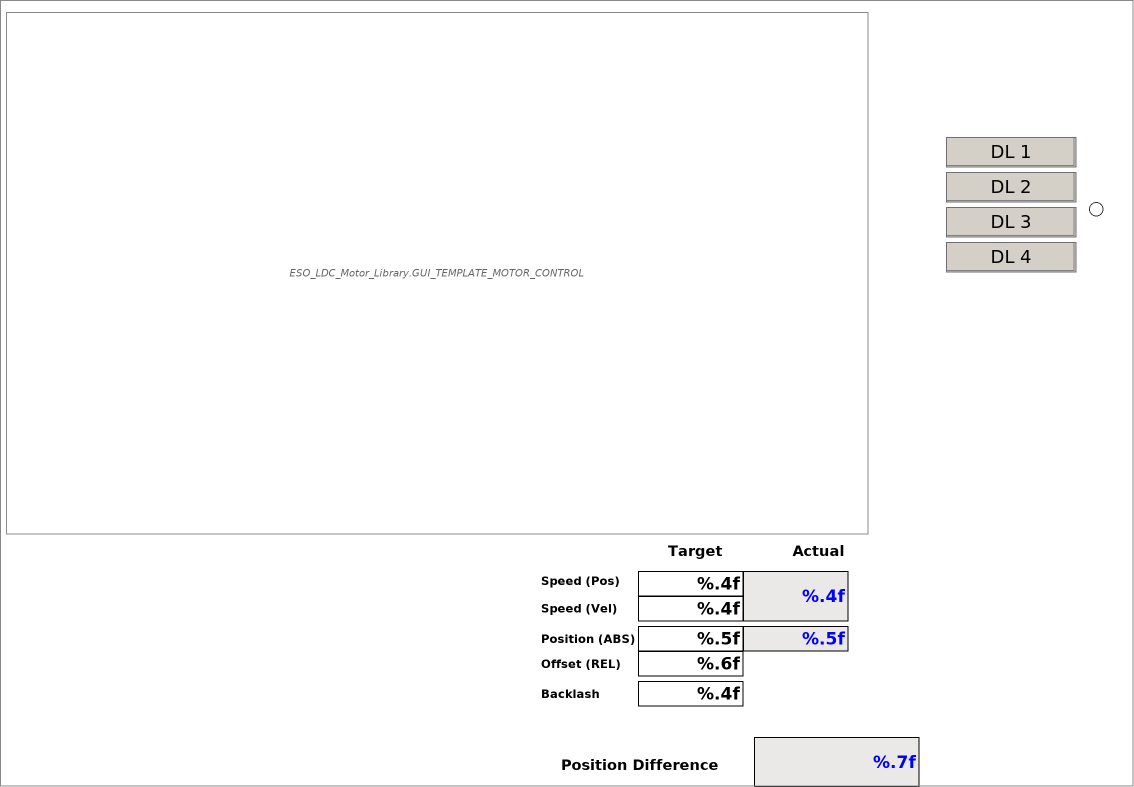
VISUALIZATION GUI_NOTT_DL_CTRL  // 1134x787
    RadioButton (1087,139 47x140), variable: MAIN.nott_ics.Delay_Lines.guiShutterIndex-1
        Areas[0]: Text=Radiobutton
        Areas[1]: Text=Radiobutton
    Button (946,137 130x30), "DL 1"
        OnMouseClick: execute { MAIN.nott_ics.Delay_Lines.guiShutterIndex := 1; }
    Button (946,172 130x30), "DL 2"
        OnMouseClick: execute { MAIN.nott_ics.Delay_Lines.guiShutterIndex := 2; }
    Button (946,207 130x30), "DL 3"
        OnMouseClick: execute { MAIN.nott_ics.Delay_Lines.guiShutterIndex := 3; }
    Button (946,242 130x30), "DL 4"
        OnMouseClick: execute { MAIN.nott_ics.Delay_Lines.guiShutterIndex := 4; }
    Frame (6,12 862x522)
        shows ESO_LDC_Motor_Library.GUI_TEMPLATE_MOTOR_CONTROL(m_Instance := MAIN.nott_ics.Delay_Lines.ptrDelayLines[MAIN.nott_ics.Delay_Lines.guiShutterIndex]^)
    Rectangle (538,571 95x20), "Speed (Pos)"
    Rectangle (743,626 105x25), "%.5f", text variable: MAIN.nott_ics.Delay_Lines.ptrDelayLines[MAIN.nott_ics.Delay_Lines.guiShutterIndex]^.stat.lrPosActual, input disabled if: false
    Rectangle (665,541 190x20), "Target Actual"
    Rectangle (538,629 95x20), "Position (ABS)"
    Rectangle (743,571 105x50), "%.4f", text variable: MAIN.nott_ics.Delay_Lines.ptrDelayLines[MAIN.nott_ics.Delay_Lines.guiShutterIndex]^.stat.lrVelActual, input disabled if: false
    Rectangle (638,596 105x25), "%.4f", text variable: MAIN.nott_ics.Delay_Lines.ptrDelayLines[MAIN.nott_ics.Delay_Lines.guiShutterIndex]^.ctrl.lrVelocity
        OnMouseDown: write the text variable via Default
    Rectangle (538,684 95x20), "Backlash"
    Rectangle (638,681 105x25), "%.4f", text variable: MAIN.nott_ics.Delay_Lines.ptrDelayLines[MAIN.nott_ics.Delay_Lines.guiShutterIndex]^.cfg.lrBacklash
        OnMouseDown: write the text variable via Default
    Rectangle (538,596 95x25), "Speed (Vel)"
    Rectangle (638,626 105x25), "%.5f", tooltip "Absolute position used by "MOVE ABS"", text variable: MAIN.nott_ics.Delay_Lines.ptrDelayLines[MAIN.nott_ics.Delay_Lines.guiShutterIndex]^.ctrl.lrPosition
        OnMouseDown: write the text variable via Default
    Rectangle (638,571 105x25), "%.4f", text variable: MAIN.nott_ics.Delay_Lines.ptrDelayLines[MAIN.nott_ics.Delay_Lines.guiShutterIndex]^.cfg.lrDefaultVelocity
        OnMouseDown: write the text variable via Default
    Rectangle (538,654 95x20), "Offset (REL)"
    Rectangle (638,651 105x25), "%.6f", tooltip "Relative offset used by "MOVE REL"", text variable: MAIN.nott_ics.Delay_Lines.ptrDelayLines[MAIN.nott_ics.Delay_Lines.guiShutterIndex]^.ctrl.lrOffset
        OnMouseDown: write the text variable via Default
    Rectangle (754,737 165x50), "%.7f", text variable: MAIN.nott_ics.Delay_Lines.ptrDelayLines[MAIN.nott_ics.Delay_Lines.guiShutterIndex]^.stat.lrPosError, input disabled if: false
    Rectangle (558,755 190x20), "Position Difference"
END_VISUALIZATION

// ---- VISUs/GUIs/GUI_NOTT_DL_1.TcVIS
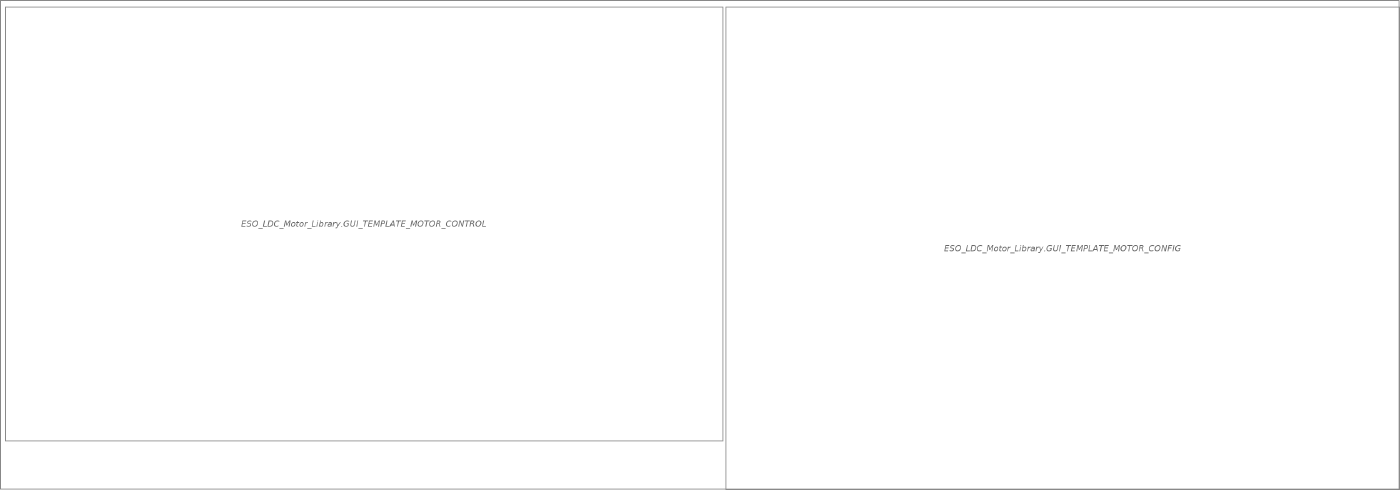
VISUALIZATION GUI_NOTT_DL_1  // 1681x589
    Frame (6,8 862x522)
        shows ESO_LDC_Motor_Library.GUI_TEMPLATE_MOTOR_CONTROL(m_Instance := MAIN.nott_ics.Delay_Lines.NDL1)
    Frame (871,8 810x581)
        shows ESO_LDC_Motor_Library.GUI_TEMPLATE_MOTOR_CONFIG(m_Instance := MAIN.nott_ics.Delay_Lines.NDL1)
END_VISUALIZATION

// ---- VISUs/GUIs/Shutters/GUI_NOTT_SHUTTERS.TcVIS
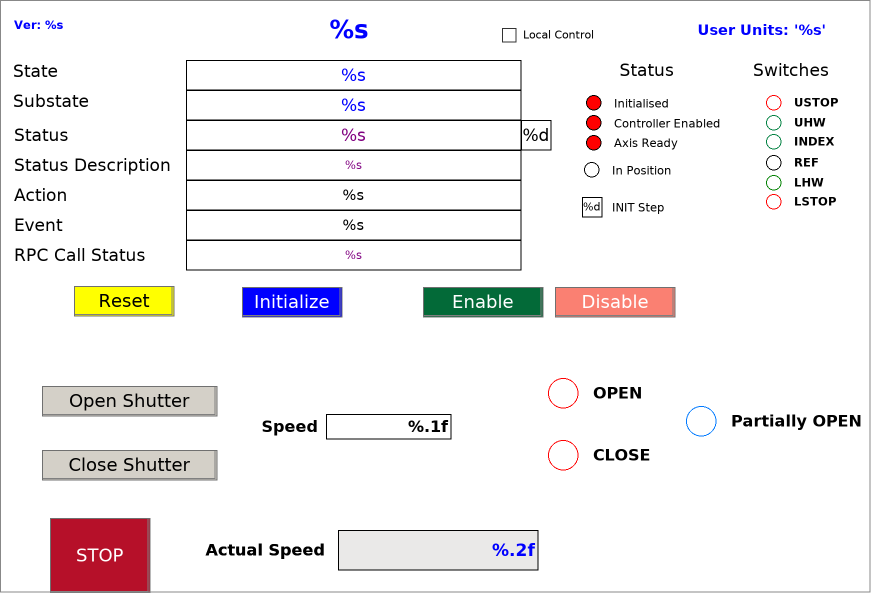
VISUALIZATION GUI_NOTT_SHUTTERS  // 871x593
    Rectangle (186,60 335x30), "%s", text variable: m_Instance.stat.sState
    Rectangle (186,90 335x30), "%s", text variable: m_Instance.stat.sSubstate
    Button (74,286 100x30), "Reset", input disabled if: NOT m_Instance.stat.bLocal OR NOT m_Instance.in_bSafe
        OnMouseDown: execute {
            m_Instance.ctrl.bLocalCmd := TRUE;
            m_Instance.ctrl.nCommand := E_MOTOR_COMMAND.RESET;
            m_Instance.ctrl.bExecute := TRUE;
        }
    Button (242,287 100x30), "Initialize", input disabled if: NOT m_Instance.stat.bLocal OR NOT m_Instance.in_bSafe
        OnMouseDown: execute {
            m_Instance.ctrl.bLocalCmd := TRUE;
            m_Instance.ctrl.nCommand := E_MOTOR_COMMAND.INIT;
            m_Instance.ctrl.bExecute := TRUE;
        }
    Button (50,518 100x75), "STOP", input disabled if: NOT m_Instance.stat.bLocal OR NOT m_Instance.in_bSafe
        OnMouseDown: execute {
            m_Instance.ctrl.bLocalCmd := TRUE;
            m_Instance.ctrl.nCommand := E_MOTOR_COMMAND.STOP;
            m_Instance.ctrl.bExecute := TRUE;
        }
    Button (423,287 120x30), "Enable", input disabled if: NOT m_Instance.stat.bLocal OR NOT m_Instance.in_bSafe
        OnMouseDown: execute {
            m_Instance.ctrl.bLocalCmd := TRUE;
            m_Instance.ctrl.nCommand := E_MOTOR_COMMAND.ENABLE;
            m_Instance.ctrl.bExecute := TRUE;
        }
    Button (555,287 120x30), "Disable", input disabled if: NOT m_Instance.stat.bLocal OR NOT m_Instance.in_bSafe
        OnMouseDown: execute {
            m_Instance.ctrl.bLocalCmd := TRUE;
            m_Instance.ctrl.nCommand := E_MOTOR_COMMAND.DISABLE;
            m_Instance.ctrl.bExecute := TRUE;
        }
    Rectangle (10,56 170x30), "State"
    Rectangle (10,86 170x30), "Substate"
    Rectangle (186,120 335x30), "%s", text variable: m_Instance.stat.sStatus
    Rectangle (186,150 335x30), "%s", tooltip "Additional information mostly used for description of errors", text variable: m_Instance.stat.sErrorText
    Rectangle (11,120 170x30), "Status"
    Rectangle (11,150 170x30), "Status Description"
    Rectangle (186,180 335x30), "%s", text variable: m_Instance.stat.sActionDesc
    Rectangle (186,210 335x30), "%s", text variable: m_Instance.stat.sEventDesc
    Rectangle (11,180 170x30), "Action"
    Rectangle (11,210 170x30), "Event"
    Rectangle (233,12 232x35), "%s", text variable: m_Instance.sName
    Checkbox (500,20 116x30), "Local Control", variable: m_Instance.stat.bLocal
    Rectangle (601,55 92x30), "Status"
    Rectangle (521,120 30x30), "%d", text variable: m_Instance.stat.nStatus
    Rectangle (745,55 92x30), "Switches"
    Rectangle (791,95 50x15), "USTOP"
    Ellipse (766,95 15x15), colour toggle: m_Instance.stat.signals[5].bActive
    Ellipse (766,115 15x15), colour toggle: m_Instance.stat.signals[4].bActive
    Ellipse (766,175 15x15), colour toggle: m_Instance.stat.signals[1].bActive
    Ellipse (766,194 15x15), colour toggle: m_Instance.stat.signals[0].bActive
    Ellipse (766,155 15x15), colour toggle: m_Instance.stat.signals[2].bActive
    Rectangle (791,134 50x15), "INDEX"
    Rectangle (791,115 50x15), "UHW"
    Rectangle (791,155 50x15), "REF"
    Rectangle (791,175 50x15), "LHW"
    Rectangle (791,194 50x15), "LSTOP"
    Ellipse (766,134 15x15), colour toggle: m_Instance.stat.signals[3].bActive
    Ellipse (586,95 15x15), tooltip "GREEN = Initialised RED = Not Initialised", text variable: m_Instance.stat.bInitialised, colour toggle: m_Instance.stat.bInitialised
    Rectangle (611,91 90x25), "Initialised"
    Rectangle (611,111 125x25), "Controller Enabled"
    Rectangle (611,131 90x24), "Axis Ready"
    Ellipse (586,115 15x15), tooltip "GREEN = Enabled RED = Disabled", colour toggle: m_Instance.stat.bEnabled
    Ellipse (586,135 15x15), tooltip "GREEN = Ready RED = Not Ready", colour toggle: m_Instance.stat.bAxisReady
    Rectangle (582,197 20x20), "%d", text variable: m_Instance.stat.nInitStep
    Rectangle (609,195 90x25), "INIT Step"
    Rectangle (11,240 170x30), "RPC Call Status"
    Rectangle (186,240 335x30), "%s", text variable: m_Instance.stat.sRPCErrorText
    Rectangle (609,158 90x25), "In Position"
    Ellipse (584,162 15x15), tooltip "GREEN = In Position BLANK = Not In Position (or not used)", colour toggle: (m_Instance.stat.bInPosition) <> 0
    Rectangle (626,15 203x30), "User Units: '%s'", text variable: m_Instance.stat.axis.sUnits
    Rectangle (11,10 99x30), "Ver: %s", tooltip "'Motor.library version'", text variable: m_Instance.stat.sLibVersion, input disabled if: true
    Group (178,530 360x40)
        Rectangle (160,0 200x40), "%.2f", text variable: m_Instance.stat.lrVelActual, input disabled if: false
        Rectangle (0,5 150x30), "Actual Speed"
    Rectangle (338,530 200x40), "%.2f", text variable: m_Instance.stat.lrVelActual, input disabled if: false
    Rectangle (178,535 150x30), "Actual Speed"
    Rectangle (226,414 95x25), "Speed", tooltip "Shutter Speed (mm/sec)"
    Rectangle (326,414 125x25), "%.1f", text variable: m_Instance.ctrl.lrVelocity
        OnMouseDown: write the text variable via Default
    Button (42,386 175x30), "Open Shutter", input disabled if: NOT m_Instance.stat.bLocal OR NOT m_Instance.in_bSafe
        OnMouseDown: execute {
            m_Instance.ctrl.bLocalCmd := TRUE;
            m_Instance.ctrl.nCommand := E_MOTOR_COMMAND.MOTOR_MOVE;
            m_Instance.ctrl.nMoveType := E_MOTOR_MOVE_TYPE.VELOCITY;
            m_Instance.ctrl.nDirection := MC_Negative_Direction;
            m_Instance.ctrl.bExecute := TRUE;
        }
    Button (42,450 175x30), "Close Shutter", input disabled if: NOT m_Instance.stat.bLocal OR NOT m_Instance.in_bSafe
        OnMouseDown: execute {
            m_Instance.ctrl.bLocalCmd := TRUE;
            m_Instance.ctrl.nCommand := E_MOTOR_COMMAND.MOTOR_MOVE;
            m_Instance.ctrl.nMoveType := E_MOTOR_MOVE_TYPE.VELOCITY;
            m_Instance.ctrl.nDirection := MC_Positive_Direction;
            m_Instance.ctrl.bExecute := TRUE;
        }
    Ellipse (548,378 30x30), colour toggle: m_Instance.stat.signals[5].bActive
    Rectangle (590,378 100x30), "OPEN", tooltip "Shutter is Open"
    Ellipse (548,440 30x30), colour toggle: m_Instance.stat.signals[0].bActive
    Rectangle (590,440 100x30), "CLOSE", tooltip "Shutter is closed"
    Ellipse (686,406 30x30), colour toggle: m_Instance.bShutterPartiallyOpen
    Rectangle (728,406 143x30), "Partially OPEN", tooltip "Either shutter is opening or closing"
END_VISUALIZATION

// ---- VISUs/GUIs/Time/GUI_NOTT_TIME.TcVIS
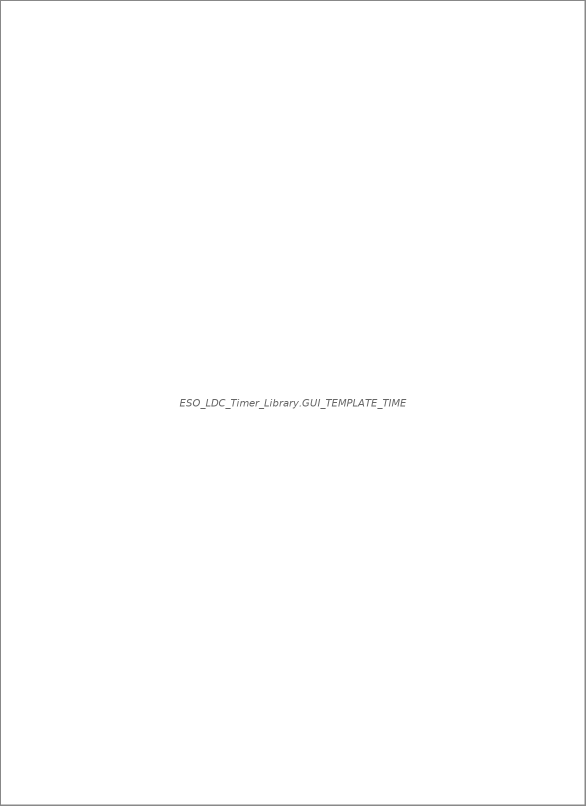
VISUALIZATION GUI_NOTT_TIME  // 586x806
    Frame (0,0 586x806)
        shows ESO_LDC_Timer_Library.GUI_TEMPLATE_TIME(m_DeviceName := 'NOTT Time', m_Instance := INFRATEC_TRIGERS.NottTime)
END_VISUALIZATION

// ---- VISUs/GUIs/TipTilt/GUI_NOTT_TIP_A_CONFIG.TcVIS
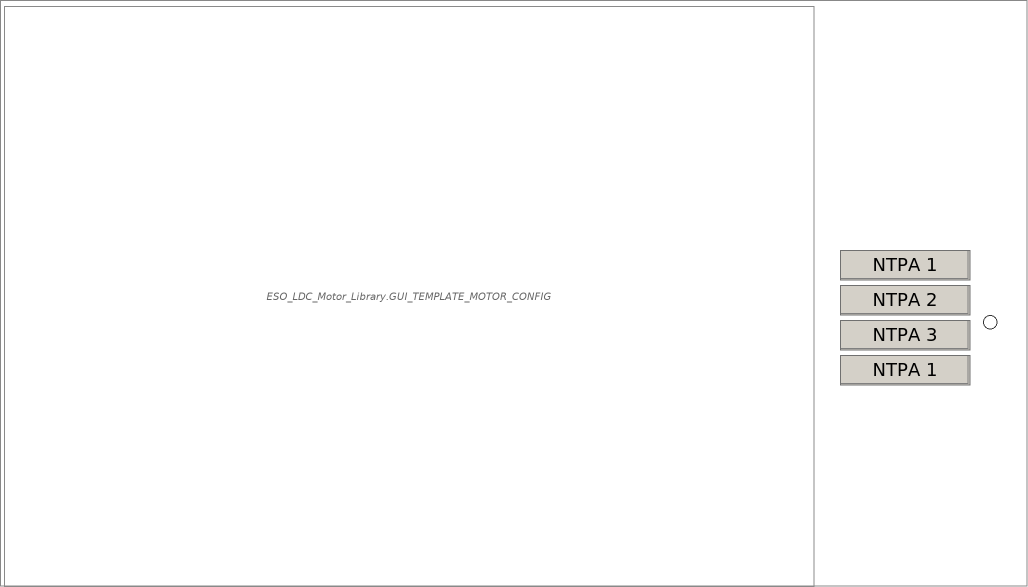
VISUALIZATION GUI_NOTT_TIP_A_CONFIG  // 1028x587
    Frame (4,6 810x581)
        shows ESO_LDC_Motor_Library.GUI_TEMPLATE_MOTOR_CONFIG(m_Instance := MAIN.nott_ics.TipTilt.ptrTipActuatorsA[MAIN.nott_ics.TipTilt.guiTipActuatorsAIndex]^)
    RadioButton (981,252 47x140), variable: MAIN.nott_ics.TipTilt.guiTipActuatorsAIndex-1
        Areas[0]: Text=Radiobutton
        Areas[1]: Text=Radiobutton
    Button (840,250 130x30), "NTPA 1"
        OnMouseClick: execute { MAIN.nott_ics.TipTilt.guiTipActuatorsAIndex := 1; }
    Button (840,285 130x30), "NTPA 2"
        OnMouseClick: execute { MAIN.nott_ics.TipTilt.guiTipActuatorsAIndex := 2; }
    Button (840,320 130x30), "NTPA 3"
        OnMouseClick: execute { MAIN.nott_ics.TipTilt.guiTipActuatorsAIndex := 3; }
    Button (840,355 130x30), "NTPA 1"
        OnMouseClick: execute { MAIN.nott_ics.TipTilt.guiTipActuatorsAIndex := 4; }
END_VISUALIZATION

// ---- VISUs/GUIs/TipTilt/GUI_NOTT_TIP_B_CONFIG.TcVIS
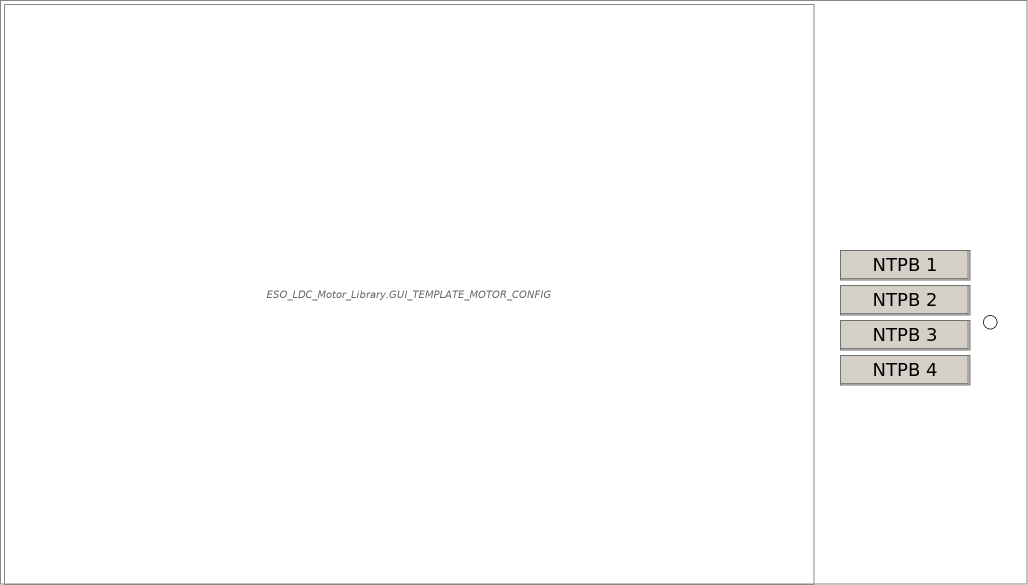
VISUALIZATION GUI_NOTT_TIP_B_CONFIG  // 1028x585
    Frame (4,4 810x581)
        shows ESO_LDC_Motor_Library.GUI_TEMPLATE_MOTOR_CONFIG(m_Instance := MAIN.nott_ics.TipTilt.ptrTipActuatorsB[MAIN.nott_ics.TipTilt.guiTipActuatorsBIndex]^)
    RadioButton (981,252 47x140), variable: MAIN.nott_ics.TipTilt.guiTipActuatorsBIndex-1
        Areas[0]: Text=Radiobutton
        Areas[1]: Text=Radiobutton
    Button (840,250 130x30), "NTPB 1"
        OnMouseClick: execute { MAIN.nott_ics.TipTilt.guiTipActuatorsBIndex := 1; }
    Button (840,285 130x30), "NTPB 2"
        OnMouseClick: execute { MAIN.nott_ics.TipTilt.guiTipActuatorsBIndex := 2; }
    Button (840,320 130x30), "NTPB 3"
        OnMouseClick: execute { MAIN.nott_ics.TipTilt.guiTipActuatorsBIndex := 3; }
    Button (840,355 130x30), "NTPB 4"
        OnMouseClick: execute { MAIN.nott_ics.TipTilt.guiTipActuatorsBIndex := 4; }
END_VISUALIZATION

// ---- VISUs/GUIs/TipTilt/GUI_NOTT_TILT_B_CONFIG.TcVIS
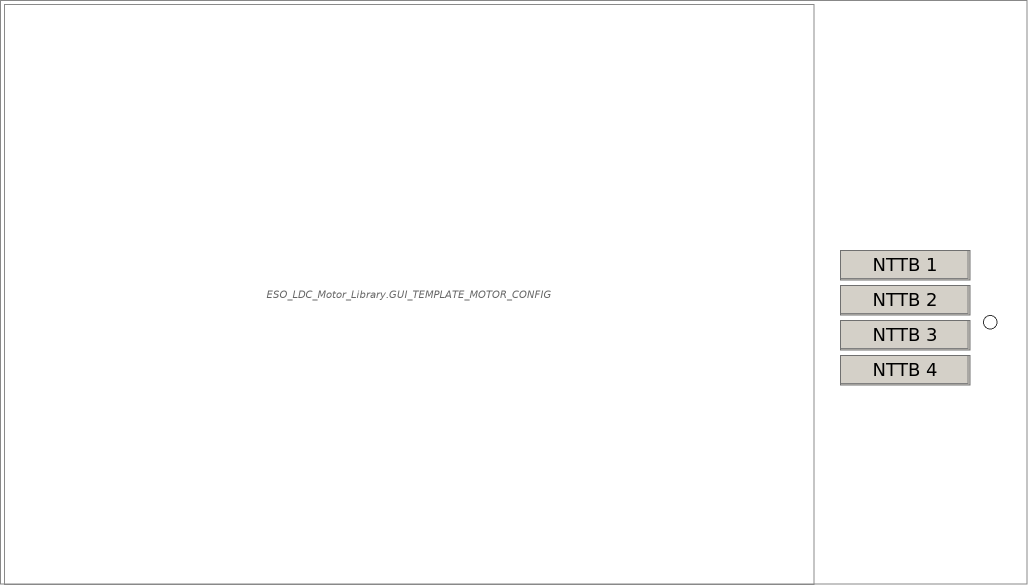
VISUALIZATION GUI_NOTT_TILT_B_CONFIG  // 1028x585
    Frame (4,4 810x581)
        shows ESO_LDC_Motor_Library.GUI_TEMPLATE_MOTOR_CONFIG(m_Instance := MAIN.nott_ics.TipTilt.ptrTiltActuatorsB[MAIN.nott_ics.TipTilt.guiTiltActuatorsBIndex]^)
    RadioButton (981,252 47x140), variable: MAIN.nott_ics.TipTilt.guiTiltActuatorsBIndex-1
        Areas[0]: Text=Radiobutton
        Areas[1]: Text=Radiobutton
    Button (840,250 130x30), "NTTB 1"
        OnMouseClick: execute { MAIN.nott_ics.TipTilt.guiTiltActuatorsBIndex := 1; }
    Button (840,285 130x30), "NTTB 2"
        OnMouseClick: execute { MAIN.nott_ics.TipTilt.guiTiltActuatorsBIndex := 2; }
    Button (840,320 130x30), "NTTB 3"
        OnMouseClick: execute { MAIN.nott_ics.TipTilt.guiTiltActuatorsBIndex := 3; }
    Button (840,355 130x30), "NTTB 4"
        OnMouseClick: execute { MAIN.nott_ics.TipTilt.guiTiltActuatorsBIndex := 4; }
END_VISUALIZATION

// ---- VISUs/GUIs/TipTilt/GUI_NOTT_TILT_A_CONFIG.TcVIS
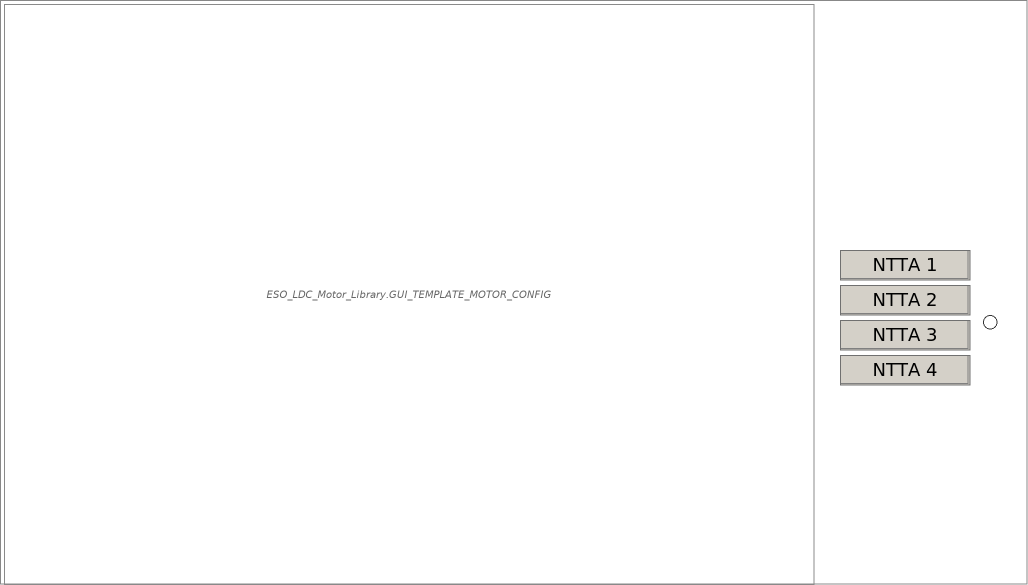
VISUALIZATION GUI_NOTT_TILT_A_CONFIG  // 1028x585
    Frame (4,4 810x581)
        shows ESO_LDC_Motor_Library.GUI_TEMPLATE_MOTOR_CONFIG(m_Instance := MAIN.nott_ics.TipTilt.ptrTiltActuatorsA[MAIN.nott_ics.TipTilt.guiTiltActuatorsAIndex]^)
    RadioButton (981,252 47x140), variable: MAIN.nott_ics.TipTilt.guiTiltActuatorsAIndex-1
        Areas[0]: Text=Radiobutton
        Areas[1]: Text=Radiobutton
    Button (840,250 130x30), "NTTA 1"
        OnMouseClick: execute { MAIN.nott_ics.TipTilt.guiTiltActuatorsAIndex := 1; }
    Button (840,285 130x30), "NTTA 2"
        OnMouseClick: execute { MAIN.nott_ics.TipTilt.guiTiltActuatorsAIndex := 2; }
    Button (840,320 130x30), "NTTA 3"
        OnMouseClick: execute { MAIN.nott_ics.TipTilt.guiTiltActuatorsAIndex := 3; }
    Button (840,355 130x30), "NTTA 4"
        OnMouseClick: execute { MAIN.nott_ics.TipTilt.guiTiltActuatorsAIndex := 4; }
END_VISUALIZATION

// ---- VISUs/GUIs/TipTilt/GUI_NOTT_TIP_A_CTRL.TcVIS
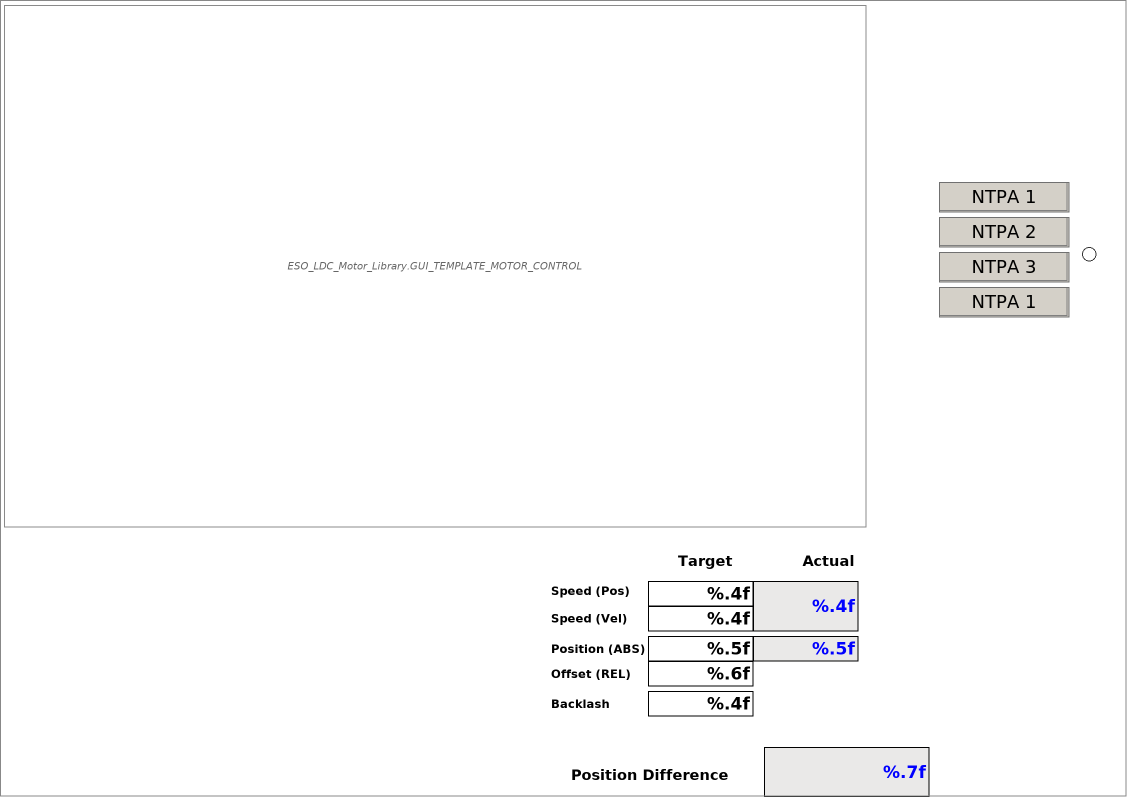
VISUALIZATION GUI_NOTT_TIP_A_CTRL  // 1127x797
    Frame (4,5 862x522)
        shows ESO_LDC_Motor_Library.GUI_TEMPLATE_MOTOR_CONTROL(m_Instance := MAIN.nott_ics.TipTilt.ptrTipActuatorsA[MAIN.nott_ics.TipTilt.guiTipActuatorsAIndex]^)
    Rectangle (548,581 95x20), "Speed (Pos)"
    Rectangle (753,636 105x25), "%.5f", text variable: MAIN.nott_ics.Delay_Lines.ptrDelayLines[MAIN.nott_ics.Delay_Lines.guiShutterIndex]^.stat.lrPosActual, input disabled if: false
    Rectangle (675,551 190x20), "Target Actual"
    Rectangle (548,639 95x20), "Position (ABS)"
    Rectangle (753,581 105x50), "%.4f", text variable: MAIN.nott_ics.Delay_Lines.ptrDelayLines[MAIN.nott_ics.Delay_Lines.guiShutterIndex]^.stat.lrVelActual, input disabled if: false
    Rectangle (648,606 105x25), "%.4f", text variable: MAIN.nott_ics.Delay_Lines.ptrDelayLines[MAIN.nott_ics.Delay_Lines.guiShutterIndex]^.ctrl.lrVelocity
        OnMouseDown: write the text variable via Default
    Rectangle (548,694 95x20), "Backlash"
    Rectangle (648,691 105x25), "%.4f", text variable: MAIN.nott_ics.Delay_Lines.ptrDelayLines[MAIN.nott_ics.Delay_Lines.guiShutterIndex]^.cfg.lrBacklash
        OnMouseDown: write the text variable via Default
    Rectangle (548,606 95x25), "Speed (Vel)"
    Rectangle (648,636 105x25), "%.5f", tooltip "Absolute position used by "MOVE ABS"", text variable: MAIN.nott_ics.Delay_Lines.ptrDelayLines[MAIN.nott_ics.Delay_Lines.guiShutterIndex]^.ctrl.lrPosition
        OnMouseDown: write the text variable via Default
    Rectangle (648,581 105x25), "%.4f", text variable: MAIN.nott_ics.Delay_Lines.ptrDelayLines[MAIN.nott_ics.Delay_Lines.guiShutterIndex]^.cfg.lrDefaultVelocity
        OnMouseDown: write the text variable via Default
    Rectangle (548,664 95x20), "Offset (REL)"
    Rectangle (648,661 105x25), "%.6f", tooltip "Relative offset used by "MOVE REL"", text variable: MAIN.nott_ics.Delay_Lines.ptrDelayLines[MAIN.nott_ics.Delay_Lines.guiShutterIndex]^.ctrl.lrOffset
        OnMouseDown: write the text variable via Default
    Rectangle (764,747 165x50), "%.7f", text variable: MAIN.nott_ics.Delay_Lines.ptrDelayLines[MAIN.nott_ics.Delay_Lines.guiShutterIndex]^.stat.lrPosError, input disabled if: false
    Rectangle (568,765 190x20), "Position Difference"
    RadioButton (1080,184 47x140), variable: MAIN.nott_ics.TipTilt.guiTipActuatorsAIndex-1
        Areas[0]: Text=Radiobutton
        Areas[1]: Text=Radiobutton
    Button (939,182 130x30), "NTPA 1"
        OnMouseClick: execute { MAIN.nott_ics.TipTilt.guiTipActuatorsAIndex := 1; }
    Button (939,217 130x30), "NTPA 2"
        OnMouseClick: execute { MAIN.nott_ics.TipTilt.guiTipActuatorsAIndex := 2; }
    Button (939,252 130x30), "NTPA 3"
        OnMouseClick: execute { MAIN.nott_ics.TipTilt.guiTipActuatorsAIndex := 3; }
    Button (939,287 130x30), "NTPA 1"
        OnMouseClick: execute { MAIN.nott_ics.TipTilt.guiTipActuatorsAIndex := 4; }
END_VISUALIZATION

// ---- VISUs/GUIs/TipTilt/GUI_NOTT_TIP_B_CTRL.TcVIS
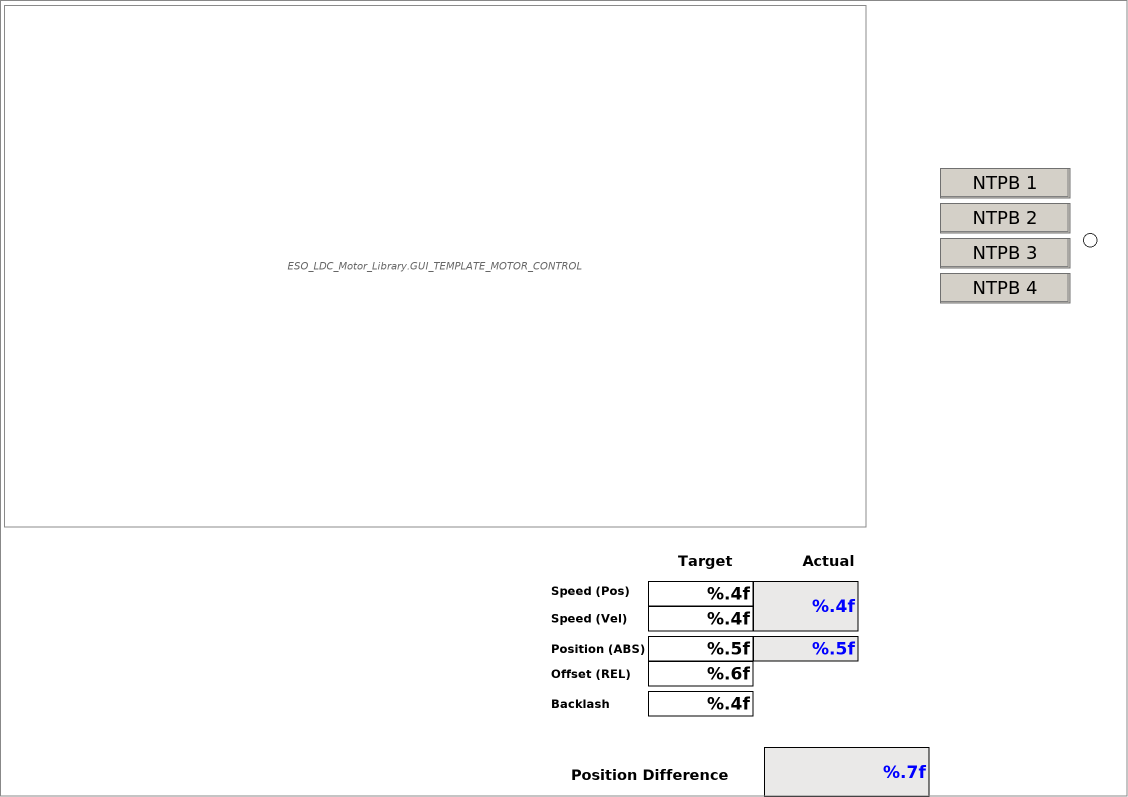
VISUALIZATION GUI_NOTT_TIP_B_CTRL  // 1128x797
    Frame (4,5 862x522)
        shows ESO_LDC_Motor_Library.GUI_TEMPLATE_MOTOR_CONTROL(m_Instance := MAIN.nott_ics.TipTilt.ptrTipActuatorsB[MAIN.nott_ics.TipTilt.guiTipActuatorsBIndex]^)
    Rectangle (548,581 95x20), "Speed (Pos)"
    Rectangle (753,636 105x25), "%.5f", text variable: MAIN.nott_ics.Delay_Lines.ptrDelayLines[MAIN.nott_ics.Delay_Lines.guiShutterIndex]^.stat.lrPosActual, input disabled if: false
    Rectangle (675,551 190x20), "Target Actual"
    Rectangle (548,639 95x20), "Position (ABS)"
    Rectangle (753,581 105x50), "%.4f", text variable: MAIN.nott_ics.Delay_Lines.ptrDelayLines[MAIN.nott_ics.Delay_Lines.guiShutterIndex]^.stat.lrVelActual, input disabled if: false
    Rectangle (648,606 105x25), "%.4f", text variable: MAIN.nott_ics.Delay_Lines.ptrDelayLines[MAIN.nott_ics.Delay_Lines.guiShutterIndex]^.ctrl.lrVelocity
        OnMouseDown: write the text variable via Default
    Rectangle (548,694 95x20), "Backlash"
    Rectangle (648,691 105x25), "%.4f", text variable: MAIN.nott_ics.Delay_Lines.ptrDelayLines[MAIN.nott_ics.Delay_Lines.guiShutterIndex]^.cfg.lrBacklash
        OnMouseDown: write the text variable via Default
    Rectangle (548,606 95x25), "Speed (Vel)"
    Rectangle (648,636 105x25), "%.5f", tooltip "Absolute position used by "MOVE ABS"", text variable: MAIN.nott_ics.Delay_Lines.ptrDelayLines[MAIN.nott_ics.Delay_Lines.guiShutterIndex]^.ctrl.lrPosition
        OnMouseDown: write the text variable via Default
    Rectangle (648,581 105x25), "%.4f", text variable: MAIN.nott_ics.Delay_Lines.ptrDelayLines[MAIN.nott_ics.Delay_Lines.guiShutterIndex]^.cfg.lrDefaultVelocity
        OnMouseDown: write the text variable via Default
    Rectangle (548,664 95x20), "Offset (REL)"
    Rectangle (648,661 105x25), "%.6f", tooltip "Relative offset used by "MOVE REL"", text variable: MAIN.nott_ics.Delay_Lines.ptrDelayLines[MAIN.nott_ics.Delay_Lines.guiShutterIndex]^.ctrl.lrOffset
        OnMouseDown: write the text variable via Default
    Rectangle (764,747 165x50), "%.7f", text variable: MAIN.nott_ics.Delay_Lines.ptrDelayLines[MAIN.nott_ics.Delay_Lines.guiShutterIndex]^.stat.lrPosError, input disabled if: false
    Rectangle (568,765 190x20), "Position Difference"
    RadioButton (1081,170 47x140), variable: MAIN.nott_ics.TipTilt.guiTipActuatorsBIndex-1
        Areas[0]: Text=Radiobutton
        Areas[1]: Text=Radiobutton
    Button (940,168 130x30), "NTPB 1"
        OnMouseClick: execute { MAIN.nott_ics.TipTilt.guiTipActuatorsBIndex := 1; }
    Button (940,203 130x30), "NTPB 2"
        OnMouseClick: execute { MAIN.nott_ics.TipTilt.guiTipActuatorsBIndex := 2; }
    Button (940,238 130x30), "NTPB 3"
        OnMouseClick: execute { MAIN.nott_ics.TipTilt.guiTipActuatorsBIndex := 3; }
    Button (940,273 130x30), "NTPB 4"
        OnMouseClick: execute { MAIN.nott_ics.TipTilt.guiTipActuatorsBIndex := 4; }
END_VISUALIZATION

// ---- VISUs/GUIs/TipTilt/GUI_NOTT_TILT_A_CTRL.TcVIS
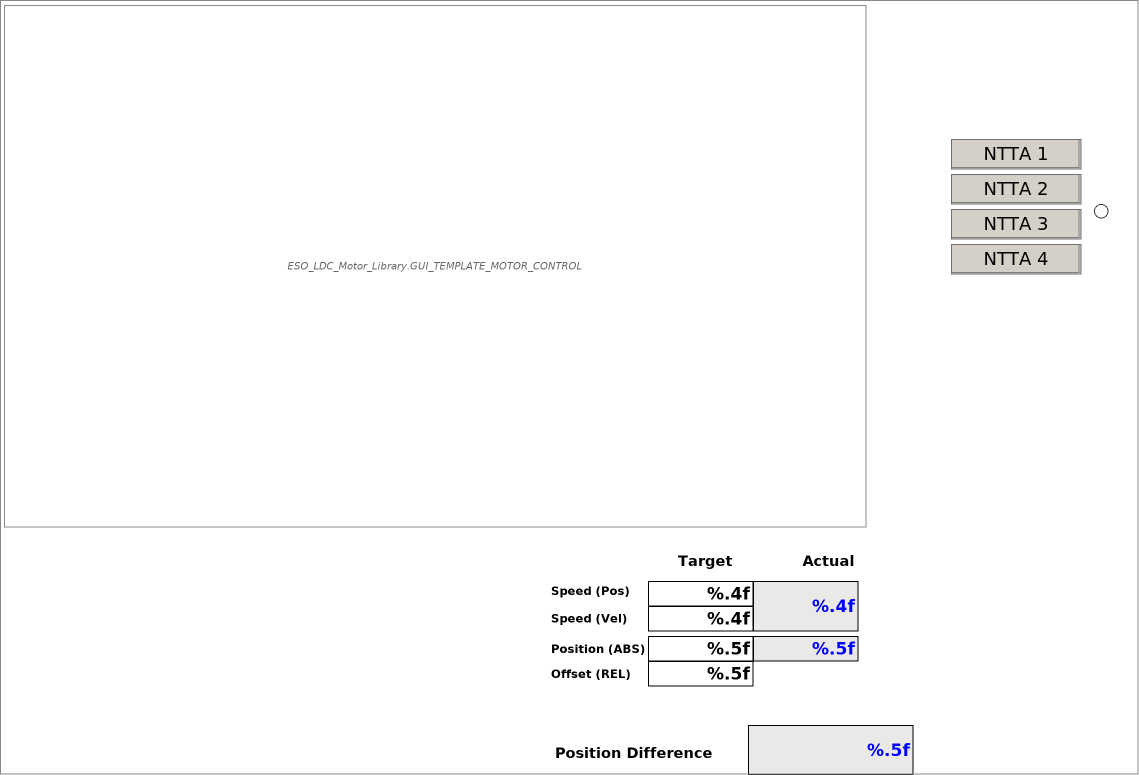
VISUALIZATION GUI_NOTT_TILT_A_CTRL  // 1139x775
    Frame (4,5 862x522)
        shows ESO_LDC_Motor_Library.GUI_TEMPLATE_MOTOR_CONTROL(m_Instance := MAIN.nott_ics.TipTilt.ptrTiltActuatorsA[MAIN.nott_ics.TipTilt.guiTiltActuatorsAIndex]^)
    Rectangle (548,581 95x20), "Speed (Pos)"
    Rectangle (753,636 105x25), "%.5f", text variable: MAIN.nott_ics.TipTilt.ptrTiltActuatorsA[MAIN.nott_ics.TipTilt.guiTiltActuatorsAIndex]^.stat.lrPosActual, input disabled if: false
    Rectangle (675,551 190x20), "Target Actual"
    Rectangle (548,639 95x20), "Position (ABS)"
    Rectangle (753,581 105x50), "%.4f", text variable: MAIN.nott_ics.TipTilt.ptrTiltActuatorsA[MAIN.nott_ics.TipTilt.guiTiltActuatorsAIndex]^.stat.lrVelActual, input disabled if: false
    Rectangle (648,606 105x25), "%.4f", text variable: MAIN.nott_ics.TipTilt.ptrTiltActuatorsA[MAIN.nott_ics.TipTilt.guiTiltActuatorsAIndex]^.ctrl.lrVelocity
        OnMouseDown: write the text variable via Default
    Rectangle (548,606 95x25), "Speed (Vel)"
    Rectangle (648,636 105x25), "%.5f", tooltip "Absolute position used by "MOVE ABS"", text variable: MAIN.nott_ics.TipTilt.ptrTiltActuatorsA[MAIN.nott_ics.TipTilt.guiTiltActuatorsAIndex]^.ctrl.lrPosition
        OnMouseDown: write the text variable via Default
    Rectangle (648,581 105x25), "%.4f", text variable: MAIN.nott_ics.TipTilt.ptrTiltActuatorsA[MAIN.nott_ics.TipTilt.guiTiltActuatorsAIndex]^.cfg.lrDefaultVelocity
        OnMouseDown: write the text variable via Default
    Rectangle (548,664 95x20), "Offset (REL)"
    Rectangle (648,661 105x25), "%.5f", tooltip "Relative offset used by "MOVE REL"", text variable: MAIN.nott_ics.TipTilt.ptrTiltActuatorsA[MAIN.nott_ics.TipTilt.guiTiltActuatorsAIndex]^.ctrl.lrOffset
        OnMouseDown: write the text variable via Default
    Rectangle (748,725 165x50), "%.5f", text variable: MAIN.nott_ics.TipTilt.ptrTiltActuatorsA[MAIN.nott_ics.TipTilt.guiTiltActuatorsAIndex]^.stat.lrPosError, input disabled if: false
    Rectangle (552,743 190x20), "Position Difference"
    RadioButton (1092,141 47x140), variable: MAIN.nott_ics.TipTilt.guiTiltActuatorsAIndex-1
        Areas[0]: Text=Radiobutton
        Areas[1]: Text=Radiobutton
    Button (951,139 130x30), "NTTA 1"
        OnMouseClick: execute { MAIN.nott_ics.TipTilt.guiTiltActuatorsAIndex := 1; }
    Button (951,174 130x30), "NTTA 2"
        OnMouseClick: execute { MAIN.nott_ics.TipTilt.guiTiltActuatorsAIndex := 2; }
    Button (951,209 130x30), "NTTA 3"
        OnMouseClick: execute { MAIN.nott_ics.TipTilt.guiTiltActuatorsAIndex := 3; }
    Button (951,244 130x30), "NTTA 4"
        OnMouseClick: execute { MAIN.nott_ics.TipTilt.guiTiltActuatorsAIndex := 4; }
END_VISUALIZATION

// ---- VISUs/GUIs/TipTilt/GUI_NOTT_TILT_B_CTRL.TcVIS
